# B&R Automation Studio project NAINV104C00R8L515F00 (part 37)

#### Act_OpsStandard_Hermes.st
```iecst
(** 2020-10-06 **)
ACTION Act_OpsStandard_Hermes:
	//InvertStepUSStandby
	//InvertStepAWMov
	IF eGotoOpsStep <> eOpsStep THEN

		CASE eGotoOpsStep OF

			ELSE
				eOpsStep	:= eGotoOpsStep;

		END_CASE

	END_IF

	Act_LogStep;

	IF eOpsStep = eGotoOpsStep THEN

		IF bPaused = FALSE THEN

			CASE eOpsStep OF

				InvertStepInitChkCondition:
					sStepTxt	:= 'Init Check Condition';

					IF p_bClampPrep THEN
						IF eInvertCurrPos	= InvertPosInvalid THEN
							bInvertPosInvalidSkipInit := TRUE;

							IF p_bClampDis THEN
								bClampDisInitUnblk	:= TRUE;
							END_IF

							eGotoOpsStep	:= InvertStepClampBlkBefInvert;
						ELSE
							eGotoOpsStep	:= InvertStepInitClampUnblk;
						END_IF
					ELSE
						IF eInvertCurrPos	= InvertPosInvalid THEN
							bInvertPosInvalidSkipInit := TRUE;

							IF (p_bInletShutterPrep AND p_bInletShutterDis=FALSE) OR (p_bOutletShutterPrep AND p_bOutletShutterDis=FALSE) THEN
								eGotoOpsStep	:= InvertStepShuttersCloseBefInvert;
							ELSE
								eGotoOpsStep	:= InvertStepInvert;
							END_IF
						ELSE
							eGotoOpsStep	:= InvertStepInitInvertComplChk;
						END_IF
					END_IF

					bPaused	:= p_bStop OR p_bStep;

				InvertStepInitClampUnblk:
					sStepTxt	:= 'Init Clamp Unblock';

					eClampAct	:= PneuActRet;

					IF p_eClampStatus = Done AND p_eClampStat = PneuActRet THEN

						eClampAct		:= PneuActIdle;
						eGotoOpsStep	:= InvertStepInitInvertComplChk;

						bPaused	:= p_bStop OR p_bStep;
					END_IF

				InvertStepInitInvertComplChk:
					sStepTxt	:= 'Init Checking Invert Complete Condition';

					IF bInvertCompl = FALSE THEN
						IF eInvertCurrPos = InvertCurrPosAtRemote THEN
							IF p_bLeftSen = TRUE THEN
								eGotoOpsStep	:= InvertStepInitConvAwayLftSen;
							ELSE
								eGotoOpsStep	:= InvertStepInitStopperBlk;
							END_IF

						ELSIF eInvertCurrPos = InvertCurrPosAtHome THEN
							IF p_bRightSen = TRUE THEN
								eGotoOpsStep	:= InvertStepInitConvAwayRgtSen;
							ELSE
								eGotoOpsStep	:= InvertStepInitStopperBlk;
							END_IF

						ELSE
							eGotoOpsStep	:= InvertStepInitStopperBlk;
						END_IF

					ELSE
						eGotoOpsStep	:= InvertStepInitStopperUnblk;
					END_IF

					bPaused	:= p_bStop OR p_bStep;

				InvertStepInitConvAwayLftSen:
					sStepTxt	:= 'Init Conveyor Away Stopper At Left';

					eConvAct	:= ConvActInit;

					fbFwdTimer(IN := TRUE, PT := DINT_TO_TIME(p_diFwdDlyTm));

					IF fbFwdTimer.Q = TRUE THEN
						fbFwdTimer(IN := FALSE);

						bHvBrd			:= FALSE;
						p_bConvHvBrd	:= FALSE;

						eConvAct		:= ConvActIdle;

						eGotoOpsStep	:= InvertStepInitStopperBlk;

						bPaused	:= p_bStop OR p_bStep;

					ELSIF p_eConvStatus = Done AND p_eConvStat = ConvActInit THEN
						fbFwdTimer(IN := FALSE);

						bHvBrd 			:= TRUE;
						bGdBrd			:= p_bInitGdBrd;

						eConvAct		:= ConvActIdle;

						eGotoOpsStep	:= InvertStepInitStopperBlk;

						bPaused	:= p_bStop OR p_bStep;
					END_IF

				InvertStepInitConvAwayRgtSen:
					sStepTxt	:= 'Init Conveyor Away Stopper At Right';

					eConvAct	:= ConvActRevImmedStart;

					fbRevTimer(IN := TRUE, PT := DINT_TO_TIME(p_diRevDlyTm));

					IF fbRevTimer.Q = TRUE THEN
						fbRevTimer(IN := FALSE);

						bHvBrd			:= FALSE;
						p_bConvHvBrd	:= FALSE;

						eConvAct		:= ConvActIdle;

						eGotoOpsStep	:= InvertStepInitStopperBlk;

						bPaused	:= p_bStop OR p_bStep;

					ELSIF p_eConvStatus = Done AND p_eConvStat = ConvActRevImmedStart THEN
						fbRevTimer(IN := FALSE);

						bHvBrd 			:= TRUE;
						bGdBrd			:= p_bInitGdBrd;

						eConvAct		:= ConvActIdle;

						eGotoOpsStep	:= InvertStepInitStopperBlk;

						bPaused	:= p_bStop OR p_bStep;
					END_IF

				InvertStepInitStopperBlk:
					sStepTxt	:= 'Init Stopper Block';

					eStopperAct	:= PneuActExt;

					IF p_eStopperStatus = Done AND p_eStopperStat = PneuActExt THEN
						eStopperAct := PneuActIdle;

						IF eInvertCurrPos = InvertCurrPosAtRemote THEN
							eGotoOpsStep  := InvertStepInitConvTwdLftSen;

						ELSIF eInvertCurrPos = InvertCurrPosAtHome THEN
							eGotoOpsStep  := InvertStepInitConvTwdRgtSen;
						END_IF

						bPaused	:= p_bStop OR p_bStep;
					END_IF

				InvertStepInitConvTwdLftSen:
					sStepTxt	:= 'Init Conveyor Toward Stopper At Left';

					eConvAct	:= ConvActRevImmedStart;

					fbRevTimer(IN := TRUE, PT := DINT_TO_TIME(p_diRevDlyTm));

					IF fbRevTimer.Q = TRUE THEN
						fbRevTimer(IN := FALSE);

						bHvBrd			:= FALSE;
						p_bConvHvBrd	:= FALSE;

						eConvAct		:= ConvActIdle;

						IF p_bClampPrep AND p_bClampDis=FALSE THEN
							eGotoOpsStep	:= InvertStepClampBlkBefInvert;
						ELSE
							IF (p_bInletShutterPrep AND p_bInletShutterDis=FALSE) OR (p_bOutletShutterPrep AND p_bOutletShutterDis=FALSE) THEN
								eGotoOpsStep	:= InvertStepShuttersCloseBefInvert;
							ELSE
								eGotoOpsStep	:= InvertStepInvert;
							END_IF
						END_IF

						bPaused	:= p_bStop OR p_bStep;

					ELSIF p_eConvStatus = Done AND p_eConvStat = ConvActRevImmedStart THEN
						fbRevTimer(IN := FALSE);
						eConvAct	:= ConvActIdle;

						bHvBrd			:= TRUE;
						bGdBrd			:= p_bInitGdBrd;

						IF p_bClampPrep AND p_bClampDis=FALSE THEN
							eGotoOpsStep	:= InvertStepClampBlkBefInvert;
						ELSE
							IF (p_bInletShutterPrep AND p_bInletShutterDis=FALSE) OR (p_bOutletShutterPrep AND p_bOutletShutterDis=FALSE) THEN
								eGotoOpsStep	:= InvertStepShuttersCloseBefInvert;
							ELSE
								eGotoOpsStep	:= InvertStepInvert;
							END_IF
						END_IF

						bPaused	:= p_bStop OR p_bStep;

					END_IF

				InvertStepInitConvTwdRgtSen:
					sStepTxt	:= 'Init Conveyor Toward Stopper at Right';

					eConvAct	:= ConvActInit;

					fbFwdTimer(IN := TRUE, PT := DINT_TO_TIME(p_diFwdDlyTm));

					IF fbFwdTimer.Q = TRUE THEN
						fbFwdTimer(IN := FALSE);

						bHvBrd			:= FALSE;
						p_bConvHvBrd	:= FALSE;

						eConvAct	:= ConvActIdle;

						IF p_bClampPrep AND p_bClampDis=FALSE THEN
							eGotoOpsStep	:= InvertStepClampBlkBefInvert;
						ELSE
							IF (p_bInletShutterPrep AND p_bInletShutterDis=FALSE) OR (p_bOutletShutterPrep AND p_bOutletShutterDis=FALSE) THEN
								eGotoOpsStep	:= InvertStepShuttersCloseBefInvert;
							ELSE
								eGotoOpsStep	:= InvertStepInvert;
							END_IF
						END_IF

						bPaused	:= p_bStop OR p_bStep;

					ELSIF p_eConvStatus = Done AND p_eConvStat = ConvActInit THEN
						fbFwdTimer(IN := FALSE);
						eConvAct	:= ConvActIdle;

						bHvBrd			:= TRUE;
						bGdBrd			:= p_bInitGdBrd;

						IF p_bClampPrep AND p_bClampDis=FALSE THEN
							eGotoOpsStep	:= InvertStepClampBlkBefInvert;
						ELSE
							IF (p_bInletShutterPrep AND p_bInletShutterDis=FALSE) OR (p_bOutletShutterPrep AND p_bOutletShutterDis=FALSE) THEN
								eGotoOpsStep	:= InvertStepShuttersCloseBefInvert;
							ELSE
								eGotoOpsStep	:= InvertStepInvert;
							END_IF
						END_IF

						bPaused	:= p_bStop OR p_bStep;
					END_IF

				InvertStepInitStopperUnblk:
					sStepTxt	:= 'Init Stopper Unblock';

					eStopperAct	:= PneuActRet;

					IF p_eStopperStatus = Done AND p_eStopperStat = PneuActRet THEN
						eStopperAct		:= PneuActIdle;
						eGotoOpsStep	:= InvertStepInitConvToRgt;

						bPaused	:= p_bStop OR p_bStep;
					END_IF

				InvertStepInitConvToRgt:
					sStepTxt	:= 'Init Conveyor to Right';

					eConvAct	:= ConvActInit;

					IF p_eConvStatus = Done AND p_eConvStat = ConvActInit THEN
						eConvAct		:= ConvActIdle;

						IF (p_bInletShutterPrep AND p_bInletShutterDis=FALSE) OR (p_bOutletShutterPrep AND p_bOutletShutterDis=FALSE) THEN
							eGotoOpsStep	:= InvertStepInitShuttersInOutClose;
						ELSE
							IF (p_bRightSen = TRUE AND NOT(p_bUSReversal)) OR (p_bLeftSen AND p_bUSReversal)   THEN //changed
								bHvBrd 	:= TRUE;
								bGdBrd	:= p_bInitGdBrd;

								eGotoOpsStep	:= InvertStepDSStandby;
							ELSE
								IF p_bAWWidthPosDiff = TRUE THEN
									eGotoOpsStep	:= InvertStepAWMov;
								ELSE
									eGotoOpsStep	:= InvertStepChkCondition;
								END_IF
							END_IF

						END_IF

						bPaused	:= p_bStop OR p_bStep;
					END_IF

				InvertStepInitShuttersInOutClose:
					sStepTxt			:= 'Init Closing Shutters';

					eInletShutterAct	:= PneuActExt;
					eOutletShutterAct	:= PneuActExt;

					IF (p_eInletShutterStatus = Done AND p_eInletShutterStat = PneuActExt) AND (p_eOutletShutterStatus = Done AND p_eOutletShutterStat = PneuActExt) THEN

						eInletShutterAct	:= PneuActIdle;
						eOutletShutterAct	:= PneuActIdle;

						IF (p_bRightSen = TRUE AND NOT(p_bUSReversal)) OR (p_bLeftSen AND p_bUSReversal)  THEN //changed

							bHvBrd 	:= TRUE;
							bGdBrd	:= p_bInitGdBrd;

							IF p_bOutletShutterOpen THEN
								eGotoOpsStep	:= InvertStepDSStandby;
							ELSE
								IF p_iHermesAction= 1 THEN
									eGotoOpsStep	:= InvertStepOutletShutterOpen;
								ELSE
									eGotoOpsStep	:= InvertStepDSInOutletShutterOpen;
								END_IF
							END_IF

						ELSE
							IF p_bAWWidthPosDiff = TRUE THEN
								eGotoOpsStep	:= InvertStepAWMov;
							ELSE
								eGotoOpsStep	:= InvertStepChkCondition;
							END_IF
						END_IF

						bPaused	:= p_bStop OR p_bStep;
					END_IF

				InvertStepShuttersInOutClose:
					sStepTxt			:= 'Closing Shutters Prior to Auto Width Change';

					eInletShutterAct	:= PneuActExt;
					eOutletShutterAct	:= PneuActExt;

					IF (p_eInletShutterStatus = Done AND p_eInletShutterStat = PneuActExt) AND (p_eOutletShutterStatus = Done AND p_eOutletShutterStat = PneuActExt) THEN

						eInletShutterAct	:= PneuActIdle;
						eOutletShutterAct	:= PneuActIdle;

						eGotoOpsStep	:= InvertStepAWMov;

						bPaused	:= p_bStop OR p_bStep;
					END_IF

				InvertStepAWMov:
					sStepTxt	:= 'Moving Auto Width';

					eAWAct	:= AWActGoWidthOff;

					IF (p_eAWStatus = Done AND p_eAWStat = AWActGoWidthOff) THEN
						eAWAct			:= AWActIdle;

						eGotoOpsStep	:= InvertStepChkCondition;

						bPaused	:= p_bStop OR p_bStep;
					END_IF

				InvertStepChkCondition:
					sStepTxt	:= 'Check Condition';

					IF (p_bInletShutterPrep AND p_bInletShutterDis=FALSE) OR (p_bOutletShutterPrep AND p_bOutletShutterDis=FALSE) THEN
						IF p_bUSAllow THEN
							eGotoOpsStep	:= InvertStepChkShutterCond;
						END_IF
					ELSE
						eGotoOpsStep	:= InvertStepStopperPosChk;
					END_IF

					bPaused	:= p_bStop OR p_bStep;

				InvertStepChkShutterCond:
					sStepTxt	:= 'Check Initial Shutter Condition';

					IF p_iHermesAction = 1 THEN
						IF p_bInletShutterOpen AND p_bOutletShutterOpen THEN//p_bOutletShutterClose THEN
							eGotoOpsStep:= InvertStepStopperPosChk;
						ELSE
							eGotoOpsStep:= InvertStepShuttersInOpenOutClose;
						END_IF
					ELSE
						IF p_bInletShutterOpen AND p_bOutletShutterOpen THEN
							eGotoOpsStep:= InvertStepStopperPosChk;
						ELSE
							eGotoOpsStep:= InvertStepShuttersInOutOpen;
						END_IF

					END_IF

					bPaused	:= p_bStop OR p_bStep;

					//Open both shutters if bypass mode
				InvertStepShuttersInOutOpen:
					sStepTxt			:= 'Opening Shutters Prior After Auto Width Change';

					eInletShutterAct	:= PneuActRet;
					eOutletShutterAct	:= PneuActRet;

					IF (p_eInletShutterStatus = Done AND p_eInletShutterStat = PneuActRet) AND (p_eOutletShutterStatus = Done AND p_eOutletShutterStat = PneuActRet) THEN

						eInletShutterAct	:= PneuActIdle;
						eOutletShutterAct	:= PneuActIdle;

						eGotoOpsStep	:= InvertStepStopperPosChk;

						bPaused	:= p_bStop OR p_bStep;
					END_IF

					//Open inlet shutter close outlet if invert mode
				InvertStepShuttersInOpenOutClose:
					sStepTxt			:= 'Opening Inlet Shutter and Closing Outlet Shutter';

					eInletShutterAct	:= PneuActRet;
					eOutletShutterAct	:= PneuActRet; //temporary testing

					IF (p_eInletShutterStatus = Done AND p_eInletShutterStat = PneuActRet) AND (p_eOutletShutterStatus = Done AND p_eOutletShutterStat = PneuActRet) THEN //PneuActExt

						eInletShutterAct	:= PneuActIdle;
						eOutletShutterAct	:= PneuActIdle;

						eGotoOpsStep	:= InvertStepStopperPosChk;

						bPaused	:= p_bStop OR p_bStep;
					END_IF

				InvertStepStopperPosChk:
					sStepTxt	:= 'Checking Stopper Position';

					IF eInvertCurrPos = InvertCurrPosAtRemote THEN
						IF NOT(p_iHermesAction = 1) THEN
							eGotoOpsStep	:= InvertStepStopperUnblk;
						ELSE
							IF NOT(p_bUSReversal) THEN
								eGotoOpsStep	:= InvertStepStopperUnblk;
							ELSE
								eGotoOpsStep	:= InvertStepStopperBlk;
							END_IF
						END_IF
					ELSIF eInvertCurrPos = InvertCurrPosAtHome THEN	//create condition if reversal
						IF NOT(p_iHermesAction = 1) THEN
							eGotoOpsStep	:= InvertStepStopperUnblk;
						ELSE
							IF NOT(p_bUSReversal) THEN
								eGotoOpsStep	:= InvertStepStopperBlk;
							ELSE
								eGotoOpsStep	:= InvertStepStopperUnblk;
							END_IF
						END_IF
					END_IF

					bPaused	:= p_bStop OR p_bStep;

				InvertStepStopperBlk:
					sStepTxt	:= 'Stopper Block';

					eStopperAct	:= PneuActExt;

					IF p_eStopperStatus = Done AND p_eStopperStat = PneuActExt THEN
						eStopperAct		:= PneuActIdle;
						eGotoOpsStep	:= InvertStepUSStandby;

						bPaused	:= p_bStop OR p_bStep;
					END_IF

				InvertStepStopperUnblk:
					sStepTxt	:= 'Stopper Unblock';

					eStopperAct	:= PneuActRet;

					IF p_eStopperStatus = Done AND p_eStopperStat = PneuActRet THEN
						eStopperAct		:= PneuActIdle;
						eGotoOpsStep	:= InvertStepUSStandby;

						bPaused	:= p_bStop OR p_bStep;
					END_IF

				InvertStepUSStandby:
					sStepTxt	:= 'In Upstream Standby Condition';

					bUSTimerRun	:= FALSE;

					bConvSen	:= p_bLeftSen OR p_bRightSen OR p_bMidSen;

					IF p_bAWWidthPosDiff = TRUE  THEN
						IF (p_bInletShutterPrep AND p_bInletShutterDis=FALSE) OR (p_bOutletShutterPrep AND p_bOutletShutterDis=FALSE) THEN
							eGotoOpsStep	:= InvertStepShuttersInOutClose;
						ELSE
							eGotoOpsStep	:= InvertStepAWMov;
						END_IF
					ELSIF p_bUSAllow = TRUE THEN
						eGotoOpsStep	:= InvertStepUSCommTmr;
					ELSIF bConvSen = TRUE THEN
						eGotoOpsStep	:= InvertStepUSTmr;
					END_IF

					bPaused	:= p_bStop OR p_bStep;

				InvertStepUSTmr:
					sStepTxt	:= 'Inserting Board By Timer';

					bConvSen	:= p_bLeftSen OR p_bRightSen OR p_bMidSen;

					fbUSTimer(IN := bConvSen);

					IF fbUSTimer.Q = TRUE THEN
						bUSTimerRun	:= TRUE;
						fbUSTimer(IN := FALSE);

						bGdBrd	:= p_bInsertGdBrd;

						IF p_iHermesAction = 1 THEN
							IF eInvertCurrPos = InvertCurrPosAtRemote THEN
								eGotoOpsStep	:= InvertStepEntToInOff;
							ELSIF eInvertCurrPos = InvertCurrPosAtHome THEN
								eGotoOpsStep	:= InvertStepEntToEnd;
							END_IF
						ELSE
							eGotoOpsStep	:= InvertStepEntToEnd;

						END_IF

					ELSIF bConvSen = FALSE THEN
						bUSTimerRun	:= FALSE;
						fbUSTimer(IN := FALSE);

						IF p_bAWWidthPosDiff = TRUE THEN
							IF (p_bInletShutterPrep AND p_bInletShutterDis=FALSE) OR (p_bOutletShutterPrep AND p_bOutletShutterDis=FALSE) THEN
								eGotoOpsStep	:= InvertStepShuttersInOutClose;
							ELSE
								eGotoOpsStep	:= InvertStepAWMov;
							END_IF
						ELSE
							eGotoOpsStep	:= InvertStepUSStandby;
						END_IF

					ELSE
						bPaused	:= p_bStop;

						IF bPaused = TRUE THEN
							bUSTimerRun	:= FALSE;
							fbUSTimer(IN := FALSE);

							eGotoOpsStep	:= InvertStepUSStandby;
						END_IF

					END_IF

				InvertStepUSCommTmr:
					sStepTxt	:= 'Communicating Upstream Machine';

					CASE p_eUSCommMod OF
						McSetCommModSMEMA:
							fbUSTimer(IN := p_bLeftSen OR p_bRightSen OR p_bMidSen);

							eUSSMEMAAct	:= SMEMAActRun;

							IF p_bUSSMEMATransporting = TRUE THEN
								bUSTimerRun	:= FALSE;
								fbUSTimer(IN := FALSE);

								bGdBrd			:= p_bUSSMEMAUSGdBrdRdy;

								sStepTxt		:= 'Conveyor Entering Board';

								IF p_iHermesAction = 1 THEN
									IF eInvertCurrPos = InvertCurrPosAtRemote THEN
										eGotoOpsStep	:= InvertStepEntToInOff;
									ELSIF eInvertCurrPos = InvertCurrPosAtHome THEN
										eGotoOpsStep	:= InvertStepEntToEnd;
									END_IF

								ELSE
									eGotoOpsStep	:= InvertStepEntToEnd;

								END_IF

							ELSIF fbUSTimer.Q = TRUE THEN
								bUSTimerRun	:= TRUE;
								fbUSTimer(IN := FALSE);

								bGdBrd	:= p_bInsertGdBrd;

								IF p_iHermesAction = 1 THEN
									IF eInvertCurrPos = InvertCurrPosAtRemote THEN
										eGotoOpsStep	:= InvertStepEntToInOff;
									ELSIF eInvertCurrPos = InvertCurrPosAtHome THEN
										eGotoOpsStep	:= InvertStepEntToEnd;
									END_IF
								ELSE
									eGotoOpsStep	:= InvertStepEntToEnd;
								END_IF

							ELSIF (p_bAWWidthPosDiff = TRUE) OR (p_bUSAllow = FALSE) THEN
								bUSTimerRun	:= FALSE;
								fbUSTimer(IN := FALSE);

								eUSSMEMAAct	:= SMEMAActIdle;

								IF p_bAWWidthPosDiff = TRUE THEN
									IF (p_bInletShutterPrep AND p_bInletShutterDis=FALSE) OR (p_bOutletShutterPrep AND p_bOutletShutterDis=FALSE) THEN
										eGotoOpsStep	:= InvertStepShuttersInOutClose;
									ELSE
										eGotoOpsStep	:= InvertStepAWMov;
									END_IF
								ELSE
									eGotoOpsStep	:= InvertStepUSStandby;
								END_IF

							ELSE

								bPaused	:= p_bStop;

								IF bPaused = TRUE THEN
									bUSTimerRun	:= FALSE;
									fbUSTimer(IN := FALSE);

									eUSSMEMAAct	:= SMEMAActIdle;

									eGotoOpsStep	:= InvertStepUSStandby;
								END_IF

							END_IF

						McSetCommModHermes:
							fbUSTimer(IN := p_bLeftSen OR p_bRightSen OR p_bMidSen);

							IF p_bUSHermesTransporting = TRUE  THEN
								bUSTimerRun	:= FALSE;
								fbUSTimer(IN := FALSE);

								bGdBrd	:= p_bUSHermesUSGdRdy;

								IF p_iHermesAction = 1 THEN
									IF eInvertCurrPos = InvertCurrPosAtRemote THEN
										IF NOT (p_bUSReversal) THEN
											eGotoOpsStep	:= InvertStepEntToInOff;
										ELSE
											eGotoOpsStep	:= InvertStepEntToEnd;
										END_IF
									ELSIF eInvertCurrPos = InvertCurrPosAtHome THEN
										IF NOT (p_bUSReversal) THEN
											eGotoOpsStep	:= InvertStepEntToEnd;
										ELSE
											eGotoOpsStep	:= InvertStepEntToInOff;
										END_IF
									END_IF
								ELSE //when bypass + reversal then check ds allow from which sided
									IF bReverseStoppingPos THEN
										eGotoOpsStep	:= InvertStepEntToInOff;
									ELSE
										eGotoOpsStep	:= InvertStepEntToEnd;
									END_IF
								END_IF

							ELSIF fbUSTimer.Q = TRUE THEN
								bUSTimerRun	:= TRUE;
								fbUSTimer(IN := FALSE);

								bGdBrd	:= p_bInsertGdBrd;

								IF p_iHermesAction = 1 THEN
									IF eInvertCurrPos = InvertCurrPosAtRemote THEN
										IF NOT (p_bUSReversal) THEN
											eGotoOpsStep	:= InvertStepEntToInOff;
										ELSE
											eGotoOpsStep	:= InvertStepEntToEnd;
										END_IF
									ELSIF eInvertCurrPos = InvertCurrPosAtHome THEN
										IF NOT (p_bUSReversal) THEN
											eGotoOpsStep	:= InvertStepEntToEnd;
										ELSE
											eGotoOpsStep	:= InvertStepEntToInOff;
										END_IF
									END_IF
								ELSE //when bypass + reversal then
									eGotoOpsStep	:= InvertStepEntToEnd;
								END_IF

							ELSIF (p_bAWWidthPosDiff = TRUE) OR (p_bUSAllow = FALSE) THEN
								bUSTimerRun	:= FALSE;
								fbUSTimer(IN := FALSE);

								IF p_bAWWidthPosDiff = TRUE THEN
									IF (p_bInletShutterPrep AND p_bInletShutterDis=FALSE) OR (p_bOutletShutterPrep AND p_bOutletShutterDis=FALSE) THEN
										eGotoOpsStep	:= InvertStepShuttersInOutClose;
									ELSE
										eGotoOpsStep	:= InvertStepAWMov;
									END_IF
								ELSE
									eGotoOpsStep	:= InvertStepUSStandby;
								END_IF

							ELSE

								bPaused	:= p_bStop;

								IF bPaused = TRUE THEN
									bUSTimerRun	:= FALSE;
									fbUSTimer(IN := FALSE);

									eGotoOpsStep	:= InvertStepUSStandby;
								END_IF

							END_IF

					END_CASE

				InvertStepEntToEnd:
					CASE p_eUSCommMod OF
						McSetCommModSMEMA:
							IF p_bUSSMEMATransporting = FALSE AND bUSTimerRun = FALSE THEN
								eConvAct	:= ConvActStop;

								IF p_eConvStatus = Done AND p_eConvStat = ConvActStop THEN
									eConvAct		:= ConvActIdle;

									eGotoOpsStep	:= InvertStepUSStandby;

									bPaused	:= p_bStop OR p_bStep;

								END_IF

							ELSE
								IF p_bUSSMEMAConvStart OR bUSTimerRun THEN
									sStepTxt	:= 'Conveyor Entering Board';
									eConvAct	:= ConvActEnt;
								END_IF

								IF (p_bConvHvBrd = TRUE) OR bUSTimerRun THEN
									bHvBrd := TRUE;
								END_IF

								IF p_bUSSMEMAConvStop AND bUSTimerRun = FALSE THEN
									sStepTxt	:= 'Conveyor Stopping';
									eConvAct	:= ConvActStop;
								END_IF

								//Waiting Conveyor Reach End for Invert Mode
								IF p_iHermesAction = 1 THEN
									IF ((p_eUSSMEMAStatus = Done AND p_eUSSMEMAStat = SMEMAActRun) OR (bUSTimerRun = TRUE)) AND p_eConvStatus = Done AND p_eConvStat = ConvActEnt THEN
										eUSSMEMAAct		:= SMEMAActIdle;
										eGotoOpsStep	:= InvertStepInvertComplChk;

										IF p_eConvStatus <> Busy THEN
											bPaused	:= p_bStop OR p_bStep;
										END_IF
									END_IF

								ELSE
									IF (p_eUSSMEMAStatus = Done AND p_eUSSMEMAStat = SMEMAActRun) OR (bUSTimerRun = TRUE) THEN
										eUSSMEMAAct		:= SMEMAActIdle;
										eGotoOpsStep	:= InvertStepInvertComplChk;

										IF p_eConvStatus <> Busy THEN
											bPaused	:= p_bStop OR p_bStep;
										END_IF
									END_IF

								END_IF

							END_IF

						McSetCommModHermes:
							IF p_bUSHermesTransporting  OR bUSTimerRun = TRUE THEN
								sStepTxt	:= 'Conveyor Entering Board';
								eConvAct	:= ConvActEnt;
							END_IF

							IF p_bUSHermesStopTransport = TRUE AND bUSTimerRun = FALSE THEN
								sStepTxt	:= 'Conveyor Stopping';
								eConvAct	:= ConvActStop;
							END_IF

							IF (p_bConvHvBrd = TRUE) OR (bUSTimerRun = TRUE) THEN
								bHvBrd := TRUE;
							END_IF

							//Waiting Conveyor Reach End for Invert Mode
							IF p_iHermesAction = 1 THEN
								IF p_bUSHermesTransporting = FALSE OR (bUSTimerRun) THEN
									IF p_eConvStat = ConvActStop THEN
										IF p_eConvStatus = Done THEN
											eConvAct		:= ConvActIdle;
											eGotoOpsStep	:= InvertStepUSStandby;
										END_IF
									ELSE
										IF p_eConvStatus = Done AND p_eConvStat = ConvActEnt THEN
											eGotoOpsStep	:= InvertStepInvertComplChk;
										END_IF
									END_IF

									IF p_eConvStatus <> Busy THEN
										bPaused	:= p_bStop OR p_bStep;
									END_IF
								END_IF

							ELSE
								IF p_bUSHermesTransporting = FALSE OR (bUSTimerRun) THEN
									IF p_eConvStat = ConvActStop THEN
										IF p_eConvStatus = Done THEN
											eConvAct		:= ConvActIdle;
											eGotoOpsStep	:= InvertStepUSStandby;
										END_IF
									ELSE
										eGotoOpsStep	:= InvertStepInvertComplChk;
									END_IF

									IF p_eConvStatus <> Busy THEN
										bPaused	:= p_bStop OR p_bStep;
									END_IF
								END_IF

							END_IF

					END_CASE

				InvertStepEntToInOff:
					CASE p_eUSCommMod OF
						McSetCommModSMEMA:
							IF p_bUSSMEMATransporting = FALSE AND bUSTimerRun = FALSE THEN
								eConvAct	:= ConvActStop;

								IF p_eConvStatus = Done AND p_eConvStat = ConvActStop THEN
									eConvAct		:= ConvActIdle;
									eGotoOpsStep	:= InvertStepUSStandby;

									bPaused	:= p_bStop OR p_bStep;

								END_IF

							ELSE
								IF p_bUSSMEMAConvStart OR bUSTimerRun THEN
									sStepTxt	:= 'Conveyor Entering Board';
									eConvAct	:= ConvActEntToInOff;
								END_IF

								IF (p_bConvHvBrd = TRUE) OR (bUSTimerRun = TRUE) THEN
									bHvBrd := TRUE;
								END_IF

								IF p_bUSSMEMAConvStop AND bUSTimerRun = FALSE THEN
									sStepTxt	:= 'Conveyor Stopping';
									eConvAct	:= ConvActStop;
								END_IF

								IF ((p_eUSSMEMAStatus = Done AND p_eUSSMEMAStat = SMEMAActRun) OR (bUSTimerRun = TRUE)) AND p_eConvStatus = Done AND p_eConvStat = ConvActEntToInOff THEN
									eUSSMEMAAct		:= SMEMAActIdle;
									eGotoOpsStep	:= InvertStepStopperBlkAftEnt;

									IF p_eConvStatus <> Busy THEN
										bPaused	:= p_bStop OR p_bStep;
									END_IF
								END_IF

							END_IF

						McSetCommModHermes:
							IF p_bUSHermesTransporting  OR bUSTimerRun = TRUE THEN
								sStepTxt	:= 'Conveyor Entering Board';
								eConvAct	:= ConvActEntToInOff;
							END_IF

							IF p_bUSHermesStopTransport = TRUE AND bUSTimerRun = FALSE THEN
								sStepTxt	:= 'Conveyor Stopping';
								eConvAct	:= ConvActStop;
							END_IF

							IF (p_bConvHvBrd = TRUE) OR (bUSTimerRun = TRUE) THEN
								bHvBrd	:= TRUE;
							END_IF

							IF (p_bUSHermesTransporting = FALSE  OR (bUSTimerRun)) THEN
								IF p_eConvStat = ConvActStop THEN
									IF p_eConvStatus = Done THEN
										eConvAct		:= ConvActIdle;
										eGotoOpsStep	:= InvertStepUSStandby;
									END_IF
								ELSE
									IF p_eConvStatus = Done AND p_eConvStat = ConvActEntToInOff THEN
										eGotoOpsStep	:= InvertStepStopperBlkAftEnt;
									END_IF
								END_IF

								IF p_eConvStatus <> Busy THEN
									bPaused	:= p_bStop OR p_bStep;
								END_IF
							END_IF

					END_CASE

				InvertStepStopperBlkAftEnt:
					sStepTxt	:= 'Stopper Block After Entering Board';

					eStopperAct	:= PneuActExt;

					IF p_eStopperStatus = Done AND p_eStopperStat = PneuActExt THEN
						eStopperAct		:= PneuActIdle;
						eGotoOpsStep	:= InvertStepRev;

						bPaused	:= p_bStop OR p_bStep;
					END_IF

				InvertStepRev:
					sStepTxt	:= 'Conveyor Reverse Board';

					eConvAct	:= ConvActRevImmedStart;

					IF p_eConvStatus = Done AND p_eConvStat = ConvActRevImmedStart THEN
						eConvAct		:= ConvActIdle;

						eGotoOpsStep	:= InvertStepInvertComplChk;

						bPaused	:= p_bStop OR p_bStep;
					END_IF

				InvertStepInvertComplChk:
					sStepTxt		:= 'Checking Invert Complete Condition';

					IF eInvertCurrPos <> eInvertReqPos THEN
						IF p_bClampPrep AND p_bClampDis=FALSE THEN
							eGotoOpsStep	:= InvertStepClampBlkBefInvert;
						ELSE
							IF (p_bInletShutterPrep AND p_bInletShutterDis=FALSE) OR (p_bOutletShutterPrep AND p_bOutletShutterDis=FALSE) THEN
								eGotoOpsStep	:= InvertStepShuttersCloseBefInvert;
							ELSE
								eGotoOpsStep	:= InvertStepInvert;
							END_IF
						END_IF
					ELSE
						IF (p_bInletShutterPrep AND p_bInletShutterDis=FALSE) OR (p_bOutletShutterPrep AND p_bOutletShutterDis=FALSE) THEN
							IF p_bOutletShutterOpen THEN
								eGotoOpsStep	:= InvertStepDSStandby;
							ELSE
								eGotoOpsStep	:= InvertStepOutletShutterOpen;
							END_IF
						ELSE //standby on right or left sensor ?
							eGotoOpsStep	:= InvertStepDSStandby;
						END_IF
					END_IF

					IF p_eConvStatus <> Busy THEN
						bPaused	:= p_bStop OR p_bStep;
					END_IF

				InvertStepClampBlkBefInvert:
					sStepTxt	:= 'Clamp Block Prior to Inversion';

					eClampAct	:= PneuActExt;

					IF p_eClampStatus = Done AND p_eClampStat = PneuActExt THEN

						eClampAct		:= PneuActIdle;

						IF (p_bInletShutterPrep AND p_bInletShutterDis=FALSE) OR (p_bOutletShutterPrep AND p_bOutletShutterDis=FALSE) THEN
							eGotoOpsStep	:= InvertStepShuttersCloseBefInvert;
						ELSE
							eGotoOpsStep	:= InvertStepInvert;
						END_IF

						bPaused	:= p_bStop OR p_bStep;
					END_IF

				InvertStepShuttersCloseBefInvert:
					sStepTxt			:= 'Closing Shutters Prior to Inversion';

					eInletShutterAct	:= PneuActExt;
					eOutletShutterAct	:= PneuActExt;

					IF (p_eInletShutterStatus = Done AND p_eInletShutterStat = PneuActExt) AND (p_eOutletShutterStatus = Done AND p_eOutletShutterStat = PneuActExt) THEN

						eInletShutterAct	:= PneuActIdle;
						eOutletShutterAct	:= PneuActIdle;

						eGotoOpsStep	:= InvertStepInvert;

						bPaused	:= p_bStop OR p_bStep;
					END_IF

				InvertStepInvert:
					sStepTxt	:= 'Inverter Turning';

					IF eInvertReqPos = InvertCurrPosAtRemote THEN
						eInvertAct	:= MotorBrkActCW;
					ELSIF eInvertReqPos = InvertCurrPosAtHome THEN
						eInvertAct	:= MotorBrkActCCW;
					END_IF

					IF p_eInvertStatus = Done AND (p_eInvertStat = MotorBrkActCW OR p_eInvertStat = MotorBrkActCCW)THEN
						eInvertAct		:= MotorBrkActIdle;

						IF (p_bClampPrep AND p_bClampDis=FALSE) OR bClampDisInitUnblk THEN

							bClampDisInitUnblk	:= FALSE;

							eGotoOpsStep	:= InvertStepClampUnblkAftInvert;

						ELSE
							IF eInvertCurrPos = InvertCurrPosAtRemote THEN

								IF bInvertPosInvalidSkipInit THEN
									eGotoOpsStep	:= InvertStepInvalidPosRecoverBrd;
								ELSE
									IF p_bLeftSen = TRUE THEN
										eGotoOpsStep	:= InvertStepPreExit;
									ELSE
										eGotoOpsStep	:= InvertStepChkCondition;
									END_IF
								END_IF

							ELSIF eInvertCurrPos = InvertCurrPosAtHome THEN

								IF bInvertPosInvalidSkipInit THEN
									eGotoOpsStep	:= InvertStepInvalidPosRecoverBrd;
								ELSE
									IF p_bRightSen = TRUE THEN
										eGotoOpsStep	:= InvertStepStopperUnblkAftInvert;
									ELSE
										eGotoOpsStep	:= InvertStepChkCondition;
									END_IF
								END_IF
							END_IF
						END_IF

						bPaused	:= p_bStop OR p_bStep;
					END_IF

				InvertStepClampUnblkAftInvert:
					sStepTxt	:= 'Clamp Unblock After Invert';

					eClampAct	:= PneuActRet;

					IF p_eClampStatus = Done AND p_eClampStat = PneuActRet THEN
						eClampAct		:= PneuActIdle;

						IF eInvertCurrPos = InvertCurrPosAtRemote THEN

							IF bInvertPosInvalidSkipInit THEN
								eGotoOpsStep	:= InvertStepInvalidPosRecoverBrd;
							ELSE
								IF p_bLeftSen = TRUE THEN
									eGotoOpsStep	:= InvertStepPreExit;
								ELSE
									eGotoOpsStep	:= InvertStepChkCondition;
								END_IF
							END_IF

						ELSIF eInvertCurrPos = InvertCurrPosAtHome THEN

							IF bInvertPosInvalidSkipInit THEN
								eGotoOpsStep	:= InvertStepInvalidPosRecoverBrd;
							ELSE
								IF p_bRightSen = TRUE THEN
									eGotoOpsStep	:= InvertStepStopperUnblkAftInvert;
								ELSE
									eGotoOpsStep	:= InvertStepChkCondition;
								END_IF
							END_IF
						END_IF

						bPaused	:= p_bStop OR p_bStep;

					END_IF

				InvertStepInvalidPosRecoverBrd:
					sStepTxt		:= 'Conveyor Recovering Board Status';

					eConvAct	:= ConvActInit;

					IF p_eConvStatus = Done AND p_eConvStat = ConvActInit THEN
						eConvAct		:= ConvActIdle;

						IF (p_bRightSen = TRUE AND NOT(p_bUSReversal)) OR (p_bLeftSen AND p_bUSReversal) THEN //changed
							bHvBrd := TRUE;
							bGdBrd			:= p_bInitGdBrd;

							bInvertPosInvalidSkipInit := FALSE;

							IF eInvertCurrPos = InvertCurrPosAtRemote THEN
								IF (p_bInletShutterPrep AND p_bInletShutterDis=FALSE) OR (p_bOutletShutterPrep AND p_bOutletShutterDis=FALSE) THEN
									IF p_bOutletShutterOpen THEN
										eGotoOpsStep	:= InvertStepDSStandby;
									ELSE
										eGotoOpsStep	:= InvertStepOutletShutterOpen;
									END_IF
								ELSE
									eGotoOpsStep	:= InvertStepDSStandby;
								END_IF
							ELSIF eInvertCurrPos = InvertCurrPosAtHome THEN
								eGotoOpsStep	:= InvertStepStopperUnblkAftInvert;
							END_IF

						ELSE
							bInvertPosInvalidSkipInit := FALSE;
							eGotoOpsStep	:= InvertStepChkCondition;
						END_IF

						bPaused	:= p_bStop OR p_bStep;
					END_IF

				InvertStepStopperUnblkAftInvert:
					sStepTxt	:= 'Stopper Unblock After Invert';

					eStopperAct	:= PneuActRet;

					IF p_eStopperStatus = Done AND p_eStopperStat = PneuActRet THEN
						eStopperAct		:= PneuActIdle;

						IF (p_bInletShutterPrep AND p_bInletShutterDis=FALSE) OR (p_bOutletShutterPrep AND p_bOutletShutterDis=FALSE) THEN
							IF p_bOutletShutterOpen THEN
								eGotoOpsStep	:= InvertStepDSStandby;
							ELSE
								eGotoOpsStep	:= InvertStepOutletShutterOpen;
							END_IF
						ELSE
							eGotoOpsStep	:= InvertStepDSStandby;
						END_IF

						bPaused	:= p_bStop OR p_bStep;
					END_IF

				InvertStepPreExit:
					sStepTxt		:= 'Conveyor Pre-Exiting Board';

					eConvAct	:= ConvActPreExit;

					IF p_eConvStatus = Done AND p_eConvStat = ConvActPreExit THEN
						eConvAct		:= ConvActIdle;

						IF (p_bInletShutterPrep AND p_bInletShutterDis=FALSE) OR (p_bOutletShutterPrep AND p_bOutletShutterDis=FALSE) THEN
							IF p_bOutletShutterOpen THEN
								eGotoOpsStep	:= InvertStepDSStandby;
							ELSE
								eGotoOpsStep	:= InvertStepOutletShutterOpen;
							END_IF
						ELSE
							eGotoOpsStep	:= InvertStepDSStandby;
						END_IF

						bPaused	:= p_bStop OR p_bStep;
					END_IF

				InvertStepDSInOutletShutterOpen:
					sStepTxt	:= 'DS: Opening Inlet & Outlet Shutter';

					eInletShutterAct	:= PneuActRet;
					eOutletShutterAct	:= PneuActRet;

					IF (p_eInletShutterStatus = Done AND p_eInletShutterStat = PneuActRet)
						AND (p_eOutletShutterStatus = Done AND p_eOutletShutterStat = PneuActRet)THEN

						eInletShutterAct	:= PneuActIdle;
						eOutletShutterAct	:= PneuActIdle;

						eGotoOpsStep	:= InvertStepDSStandby;

						bPaused	:= p_bStop OR p_bStep;
					END_IF

				InvertStepOutletShutterOpen:
					sStepTxt	:= 'Opening Outlet Shutter';

					eOutletShutterAct	:= PneuActRet;

					IF p_eOutletShutterStatus = Done AND p_eOutletShutterStat = PneuActRet THEN
						eOutletShutterAct	:= PneuActIdle;

						eGotoOpsStep	:= InvertStepDSStandby;

						bPaused	:= p_bStop OR p_bStep;
					END_IF

				InvertStepDSStandby:
					sStepTxt	:= 'In Downstream Standby Condition';

					bDSTimerRun	:= FALSE;

					IF p_bUSReversal THEN//p_eConvDirection = ConvDirLToL OR p_eConvDirection = ConvDirRToL THEN //tight with ds reversal
						bConvSen	:= p_bLeftSen;
					ELSE
						bConvSen	:= p_bRightSen;
					END_IF

					IF bConvSen = TRUE OR p_eConvStatus <> Busy THEN
						bReachedEnd	:= TRUE;
					END_IF

					IF p_bDBAOnRgtSen THEN
						IF p_bDSAllow = TRUE AND bReachedEnd = TRUE THEN
							bReachedEnd		:= FALSE;
							eGotoOpsStep	:= InvertStepDSCommTmr;
						ELSIF (bReachedEnd = TRUE) AND (bConvSen = FALSE) THEN
							bReachedEnd		:= FALSE;
							eGotoOpsStep	:= InvertStepDSTmr;
						END_IF
					ELSE
						IF p_bDSAllow = TRUE THEN
							bReachedEnd		:= FALSE;
							eGotoOpsStep	:= InvertStepDSCommTmr;
						ELSIF (bReachedEnd = TRUE) AND (bConvSen = FALSE) THEN
							bReachedEnd		:= FALSE;
							eGotoOpsStep	:= InvertStepDSTmr;
						END_IF
					END_IF

					IF p_eConvStatus <> Busy THEN
						bPaused	:= p_bStop OR p_bStep;
					END_IF

				InvertStepDSTmr:
					sStepTxt	:= 'Removing Board By Timer';

					IF p_bUSReversal THEN// p_eConvDirection = ConvDirLToL OR p_eConvDirection = ConvDirRToL THEN
						bConvSen	:= p_bLeftSen;
					ELSE
						bConvSen	:= p_bRightSen;
					END_IF

					fbDSTimer(IN := NOT bConvSen);

					IF fbDSTimer.Q = TRUE THEN
						bDSTimerRun		:= TRUE;
						fbDSTimer(IN := FALSE);

						bHvBrd := FALSE;

						eConvAct		:= ConvActIdle;

						eGotoOpsStep	:= InvertStepChkCondition;

					ELSIF bConvSen = TRUE THEN
						bDSTimerRun		:= FALSE;
						fbDSTimer(IN := FALSE);

						eGotoOpsStep	:= InvertStepDSStandby;

					ELSE
						IF p_eConvStatus <> Busy THEN
							bPaused	:= p_bStop;

							IF bPaused = TRUE THEN
								bDSTimerRun	:= FALSE;
								fbDSTimer(IN := FALSE);
							END_IF
						END_IF

					END_IF

				InvertStepDSCommTmr:
					sStepTxt	:= 'Communicating Downstream Machine';

					IF p_bUSReversal THEN// p_eConvDirection = ConvDirLToL OR p_eConvDirection = ConvDirRToL THEN
						IF p_bLeftSen = TRUE OR p_eConvStatus <> Busy THEN
							bReachedEnd	:= TRUE;
						END_IF

						IF bReachedEnd = TRUE THEN
							fbDSTimer(IN := NOT p_bLeftSen);
						END_IF
					ELSE
						IF p_bRightSen = TRUE OR p_eConvStatus <> Busy THEN
							bReachedEnd	:= TRUE;
						END_IF

						IF bReachedEnd = TRUE THEN
							fbDSTimer(IN := NOT p_bRightSen);
						END_IF
					END_IF

					CASE p_eDSCommMod OF
						McSetCommModSMEMA:
							eDSSMEMAAct	:= SMEMAActRun;

							IF p_bDSSMEMAConvStart = TRUE THEN
								bDSTimerRun	:= FALSE;
								fbDSTimer(IN := FALSE);

								bReachedEnd	:= FALSE;

								eGotoOpsStep	:= InvertStepExitBrd;

							ELSIF fbDSTimer.Q = TRUE THEN
								bDSTimerRun		:= TRUE;
								fbDSTimer(IN := FALSE);
								bHvBrd := FALSE;

								bReachedEnd		:= FALSE;
								eDSSMEMAAct		:= SMEMAActIdle;
								eConvAct		:= ConvActIdle;

								eGotoOpsStep	:= InvertStepChkCondition;

							ELSIF p_bDSAllow = FALSE THEN
								bDSTimerRun		:= FALSE;
								fbDSTimer(IN := FALSE);

								bReachedEnd		:= FALSE;
								eDSSMEMAAct		:= SMEMAActIdle;
								eConvAct		:= ConvActIdle;

								eGotoOpsStep	:= InvertStepDSStandby;

							ELSE
								IF p_eConvStatus <> Busy THEN
									bPaused	:= p_bStop;

									IF bPaused = TRUE THEN
										fbDSTimer(IN := FALSE);

										eDSSMEMAAct	:= SMEMAActIdle;
									END_IF
								END_IF

							END_IF

						McSetCommModHermes:
							IF p_bDSHermesTransporting = TRUE THEN
								bDSTimerRun	:= FALSE;
								fbDSTimer(IN := FALSE);

								bReachedEnd	:= FALSE;

								eGotoOpsStep	:= InvertStepExitBrd;

							ELSIF fbDSTimer.Q = TRUE THEN
								bDSTimerRun	:= TRUE;
								fbDSTimer(IN := FALSE);
								bHvBrd := FALSE;

								bReachedEnd	:= FALSE;
								eConvAct		:= ConvActIdle;

								eGotoOpsStep	:= InvertStepChkCondition;

							ELSIF p_bDSAllow = FALSE THEN
								bDSTimerRun	:= FALSE;
								fbDSTimer(IN := FALSE);

								bReachedEnd	:= FALSE;

								eGotoOpsStep	:= InvertStepDSStandby;

							ELSE
								IF p_eConvStatus <> Busy THEN
									bPaused	:= p_bStop;

									IF bPaused = TRUE THEN
										fbDSTimer(IN := FALSE);
									END_IF
								END_IF

							END_IF

					END_CASE

				InvertStepExitBrd:
					CASE p_eDSCommMod OF
						McSetCommModSMEMA:
							eConvAct	:= ConvActExit;

							IF ((p_eDSSMEMAStatus = Done AND p_eDSSMEMAStat = SMEMAActRun) OR (bDSTimerRun)) AND (p_eConvStatus = Done AND p_eConvStat = ConvActExit) THEN

								eDSSMEMAAct		:= SMEMAActIdle;
								eConvAct		:= ConvActIdle;

								bHvBrd := FALSE;
								p_bConvHvBrd := FALSE;
								eGotoOpsStep	:= InvertStepChkCondition;

								bPaused	:= p_bStop OR p_bStep;

							END_IF

						McSetCommModHermes:
							eConvAct := ConvActExit;

							IF ((p_bDSHermesTransporting = FALSE) OR (bDSTimerRun)) AND (p_eConvStatus = Done AND p_eConvStat = ConvActExit) THEN
								eConvAct := ConvActIdle;

								bHvBrd := FALSE;
								p_bConvHvBrd := FALSE;

								eGotoOpsStep := InvertStepChkCondition;

								bPaused := p_bStop OR p_bStep;
							END_IF

					END_CASE

			END_CASE

		END_IF

	END_IF

	//Board Inserted/Removed
	bBrdInserted		:= bUSTimerRun;
	bBrdRemoved			:= bDSTimerRun;

	//Operation Step Status
	IF (eOpsStep = InvertStepInitConvAwayLftSen) OR (eOpsStep = InvertStepInitConvAwayRgtSen) OR (eOpsStep = InvertStepInitConvTwdLftSen) OR (eOpsStep = InvertStepInitConvTwdRgtSen) OR (eOpsStep = InvertStepInitConvToRgt) THEN
		bStepInitConv	:= TRUE;
	ELSE
		bStepInitConv	:= FALSE;
	END_IF

	bStepInitAwayStopper		:= (eOpsStep = InvertStepInitConvAwayLftSen) OR (eOpsStep = InvertStepInitConvAwayRgtSen);
	bStepInitTwdStopper			:= (eOpsStep = InvertStepInitConvTwdLftSen) OR (eOpsStep = InvertStepInitConvTwdRgtSen);
	bStepInitDone				:= (eOpsStep > InvertStepInitShuttersInOutClose) AND bInvertPosInvalidSkipInit=FALSE;
	bStepUSStandby				:= eOpsStep = InvertStepUSStandby;
	bStepUSCommTmr				:= eOpsStep = InvertStepUSCommTmr;
	bStepEntToEnd				:= eOpsStep = InvertStepEntToEnd;
	bStepEntToInOff				:= eOpsStep = InvertStepEntToInOff;
	bStepRev					:= eOpsStep = InvertStepRev;
	bStepPreExit				:= eOpsStep = InvertStepPreExit;
	bStepDSStandby				:= eOpsStep = InvertStepDSStandby;
	bStepDSCommTmr				:= eOpsStep = InvertStepDSCommTmr;
	bStepExitBrd				:= eOpsStep = InvertStepExitBrd;
	bStepInvert					:= eOpsStep = InvertStepInvert;
	bStepAWMov					:= eOpsStep = InvertStepAWMov;
END_ACTION
```

#### InputRef.var - Do Not Change!!!
```iecst
(*2020-10-06*)
(**)
(*General*)
VAR
	p_udiRstErr : REFERENCE TO UDINT;
	p_bEn : REFERENCE TO BOOL;
	p_bDis : REFERENCE TO BOOL;
	p_bRun : REFERENCE TO BOOL;
	p_bStop : REFERENCE TO BOOL;
	p_bStep : REFERENCE TO BOOL;
END_VAR
(**)
VAR
	p_bInitGdBrd : REFERENCE TO BOOL;
	p_bInsertGdBrd : REFERENCE TO BOOL;
	p_eConvDirection : REFERENCE TO eConvDir;
	p_eUSCommMod : REFERENCE TO eMcSetCommMod;
	p_eDSCommMod : REFERENCE TO eMcSetCommMod;
	p_bGoToStandby : REFERENCE TO BOOL;
	p_bUSAllow : REFERENCE TO BOOL;
	p_bDSAllow : REFERENCE TO BOOL;
	p_eUSComm2Mod : REFERENCE TO eMcSetCommMod;
	p_bRtrnUSAllow : REFERENCE TO BOOL;
	p_bRtrnDSAllow : REFERENCE TO BOOL;
	p_bLeftSen : REFERENCE TO BOOL;
	p_bRightSen : REFERENCE TO BOOL;
	p_bMidSen : REFERENCE TO BOOL;
	p_bClamp2Sen : REFERENCE TO BOOL;
	p_bClamp3Sen : REFERENCE TO BOOL;
END_VAR
(**)
VAR
	p_eUSSMEMAStat : REFERENCE TO eSMEMAAction;
	p_eUSSMEMAStatus : REFERENCE TO eFBStatus;
	p_bUSSMEMATransporting : REFERENCE TO BOOL;
	p_bUSSMEMAConvStart : REFERENCE TO BOOL;
	p_bUSSMEMAConvStop : REFERENCE TO BOOL;
	p_bUSSMEMAUSRdy : REFERENCE TO BOOL;
	p_bUSSMEMAUSGdBrdRdy : REFERENCE TO BOOL;
END_VAR
(**)
VAR
	p_eUSSMEMA2Stat : REFERENCE TO eSMEMAAction;
	p_eUSSMEMA2Status : REFERENCE TO eFBStatus;
	p_bUSSMEMA2Transporting : REFERENCE TO BOOL;
	p_bUSSMEMA2ConvStart : REFERENCE TO BOOL;
	p_bUSSMEMA2ConvStop : REFERENCE TO BOOL;
	p_bUSSMEMA2USRdy : REFERENCE TO BOOL;
	p_bUSSMEMA2USGdBrdRdy : REFERENCE TO BOOL;
END_VAR
(**)
VAR
	p_eDSSMEMAStat : REFERENCE TO eSMEMAAction;
	p_eDSSMEMAStatus : REFERENCE TO eFBStatus;
	p_bDSSMEMAConvStart : REFERENCE TO BOOL;
	p_bDSSMEMAConvStop : REFERENCE TO BOOL;
	p_bDSSMEMATimer : REFERENCE TO BOOL;
	p_bDBAOnRgtSen : REFERENCE TO BOOL;
END_VAR
(**)
VAR
	p_bUSHermesTransporting : REFERENCE TO BOOL;
	p_bUSHermesStopTransport : REFERENCE TO BOOL;
	p_bUSHermesUSRdy : REFERENCE TO BOOL;
	p_bUSHermesUSGdRdy : REFERENCE TO BOOL;
END_VAR
(**)
VAR
	p_bDSHermesTransporting : REFERENCE TO BOOL;
	p_bDSHermesStopTransport : REFERENCE TO BOOL;
END_VAR
(**)
VAR
	p_eConvStat : REFERENCE TO eConvAction;
	p_eConvStatus : REFERENCE TO eFBStatus;
	p_bConvHvBrd : REFERENCE TO BOOL;
END_VAR
(**)
VAR
	p_eStopperStat : REFERENCE TO ePneuAction;
	p_eStopperStatus : REFERENCE TO eFBStatus;
	p_bStopperExtended : REFERENCE TO BOOL;
	p_bStopperRetracted : REFERENCE TO BOOL;
END_VAR
(**)
VAR
	p_eClampStat : REFERENCE TO ePneuAction;
	p_eClampStatus : REFERENCE TO eFBStatus;
END_VAR
(**)
VAR
	p_eInletShutterStat : REFERENCE TO ePneuAction;
	p_eInletShutterStatus : REFERENCE TO eFBStatus;
	p_bInletShutterOpen : REFERENCE TO BOOL;
	p_bInletShutterClose : REFERENCE TO BOOL;
END_VAR
(**)
VAR
	p_eOutletShutterStat : REFERENCE TO ePneuAction;
	p_eOutletShutterStatus : REFERENCE TO eFBStatus;
	p_bOutletShutterOpen : REFERENCE TO BOOL;
	p_bOutletShutterClose : REFERENCE TO BOOL;
END_VAR
(**)
VAR
	p_eClamp1Stat : REFERENCE TO ePneuAction;
	p_eClamp1Status : REFERENCE TO eFBStatus;
	p_bClampRS1 : REFERENCE TO BOOL;
	p_bUnClampRS1 : REFERENCE TO BOOL;
END_VAR
(**)
VAR
	p_eClamp2Stat : REFERENCE TO ePneuAction;
	p_eClamp2Status : REFERENCE TO eFBStatus;
	p_bClampRS2 : REFERENCE TO BOOL;
	p_bUnClampRS2 : REFERENCE TO BOOL;
END_VAR
(**)
VAR
	p_eClamp3Stat : REFERENCE TO ePneuAction;
	p_eClamp3Status : REFERENCE TO eFBStatus;
	p_bClampRS3 : REFERENCE TO BOOL;
	p_bUnClampRS3 : REFERENCE TO BOOL;
END_VAR
(**)
VAR
	p_eInvertStat : REFERENCE TO eMotorBrkAction;
	p_eInvertStatus : REFERENCE TO eFBStatus;
END_VAR
(**)
VAR
	p_eAWStat : REFERENCE TO eAWAction;
	p_eAWStatus : REFERENCE TO eFBStatus;
	p_bAWWidthPosDiff : REFERENCE TO BOOL;
END_VAR
(**)
VAR
	p_sProgNm : REFERENCE TO STRING[15];
	p_bNtSettingsLoadDone : REFERENCE TO BOOL;
END_VAR
(**)
VAR
	p_bClampPrep : REFERENCE TO BOOL;
	p_bClampDis : REFERENCE TO BOOL;
	p_eClampOption : REFERENCE TO eClampType;
END_VAR
(**)
VAR
	p_bInletShutterPrep : REFERENCE TO BOOL;
	p_bInletShutterDis : REFERENCE TO BOOL;
	p_bOutletShutterPrep : REFERENCE TO BOOL;
	p_bOutletShutterDis : REFERENCE TO BOOL;
END_VAR
(**)
VAR
	p_bMachineSafetyPrep : REFERENCE TO BOOL;
	p_bUnlockCovPrep : REFERENCE TO BOOL;
	p_bLinkDICoverSwitchSig2 : REFERENCE TO BOOL;
	p_bLinkUIBypsCoverSWPress1 : REFERENCE TO BOOL;
	p_bLinkDIUnlockCoverSigFromDS : REFERENCE TO BOOL;
	p_bLinkDISafetySigFromDS : REFERENCE TO BOOL;
	p_bLinkDISafetySigFromUS : REFERENCE TO BOOL;
	p_bLinkDIUnlockCoverSigFromUS : REFERENCE TO BOOL;
END_VAR
(*Route Action Hermes Operaiton*)
VAR
	p_iHermesAction : REFERENCE TO INT;
	p_bUSReversal : REFERENCE TO BOOL;
	p_bHermesEntToReversePosition : REFERENCE TO BOOL;
END_VAR
```

#### Local.var - Do Not Change!!!
```iecst
(*2020-10-06*)
(**)
(*Local Action, State & Status*)
VAR
	eStatus : eFBStatus := Idle;
	udiStatus : UDINT := 0;
	udiStatus1 : UDINT := 0;
END_VAR
(**)
(*Local Alarm*)
VAR
	tyAlmData : tyAlmDat;
	tyAlmData1 : tyAlmDat;
	a_tyAlmText : ARRAY[10000..10099] OF tyAlmTxt := [9(0),(sAlmText:='Waiting for Return PCB from Upstream 2'),(sAlmText:='Waiting for Return PCB Transfer to Downstream'),89(0)];
END_VAR
(**)
(*Local Output*)
VAR
	sStepTxt : STRING[80];
	bPaused : BOOL;
END_VAR
(**)
VAR
	bStepInitConv : BOOL;
	bStepInitAwayStopper : BOOL;
	bStepInitTwdStopper : BOOL;
	bStepInitDone : BOOL;
	bStepUSStandby : BOOL;
	bStepUSCommTmr : BOOL;
	bStepEntToEnd : BOOL;
	bStepEntToInOff : BOOL;
	bStepRev : BOOL;
	bStepPreExit : BOOL;
	bStepDSStandby : BOOL;
	bStepDSCommTmr : BOOL;
	bStepExitBrd : BOOL;
	bStepInvert : BOOL;
	bStepAWMov : BOOL;
	bStepSafeMode : BOOL;
	bBrdInserted : BOOL;
	bBrdRemoved : BOOL;
	eUSSMEMAAct : eSMEMAAction;
	eDSSMEMAAct : eSMEMAAction;
	eUSSMEMA2Act : eSMEMAAction;
	eConvAct : eConvAction;
	eStopperAct : ePneuAction;
	eInvertAct : eMotorBrkAction;
	eAWAct : eAWAction;
	eClampAct : ePneuAction;
	eInletShutterAct : ePneuAction;
	eOutletShutterAct : ePneuAction;
	eClamp1Act : ePneuAction;
	eClamp2Act : ePneuAction;
	eClamp3Act : ePneuAction;
	bInvOnceTwicePCBOut : BOOL;
	bStepInvRtrnEntToEnd : BOOL;
	bStepInvRtrnEntToInOff : BOOL;
	bStepInvRtrnUSStandby : BOOL;
	bStepInvRtrnUSCommTmr : BOOL;
END_VAR
(**)
(*Local Input*)
VAR
	udiRstErr : UDINT := 0;
	bEn : BOOL := TRUE;
	bDis : BOOL := FALSE;
	bRun : BOOL;
	bStop : BOOL;
	bStep : BOOL;
	bInletShutterPrep : BOOL;
	bInletShutterDis : BOOL;
	bOutletShutterPrep : BOOL;
	bOutletShutterDis : BOOL;
	bClampPrep : BOOL;
	bClampDis : BOOL;
	eClampOption : eClampType;
END_VAR
(**)
VAR
	bBrdOnSen : BOOL := FALSE;
	bHvBrd : BOOL;
	bGdBrd : BOOL;
	bInitGdBrd : BOOL := TRUE;
	bInsertGdBrd : BOOL := TRUE;
	eConvDirection : eConvDir;
	eUSCommMod : eMcSetCommMod;
	eDSCommMod : eMcSetCommMod;
	bGoToStandby : BOOL;
	bUSAllow : BOOL := TRUE;
	bDSAllow : BOOL := TRUE;
	bLeftSen : BOOL;
	bRightSen : BOOL;
	bMidSen : BOOL;
	bClamp2Sen : BOOL;
	bClamp3Sen : BOOL;
	bRtrnUSAllow : BOOL := TRUE;
	bRtrnDSAllow : BOOL := TRUE;
END_VAR
(**)
VAR
	eUSSMEMAStat : eSMEMAAction;
	eUSSMEMAStatus : eFBStatus;
	bUSSMEMATransporting : BOOL;
	bUSSMEMAConvStart : BOOL;
	bUSSMEMAConvStop : BOOL;
	bUSSMEMAUSRdy : BOOL;
	bUSSMEMAUSGdBrdRdy : BOOL;
END_VAR
(**)
VAR
	eDSSMEMAStat : eSMEMAAction;
	eDSSMEMAStatus : eFBStatus;
	bDSSMEMAConvStart : BOOL;
	bDSSMEMAConvStop : BOOL;
	bDSSMEMATimer : BOOL;
END_VAR
(**)
VAR
	bUSHermesTransporting : BOOL;
	bUSHermesStopTransport : BOOL;
	bUSHermesUSRdy : BOOL;
	bUSHermesUSGdRdy : BOOL;
END_VAR
(**)
VAR
	bDSHermesTransporting : BOOL;
	bDSHermesStopTransport : BOOL;
END_VAR
(**)
VAR
	eConvStat : eConvAction;
	eConvStatus : eFBStatus;
	bConvHvBrd : BOOL;
	bConvLmtSenActivated : BOOL;
END_VAR
(**)
VAR
	eStopperStat : ePneuAction;
	eStopperStatus : eFBStatus;
	bStopperExtended : BOOL;
	bStopperRetracted : BOOL;
END_VAR
(**)
VAR
	eClampStat : ePneuAction;
	eClampStatus : eFBStatus;
END_VAR
(**)
VAR
	eInletShutterStat : ePneuAction;
	eInletShutterStatus : eFBStatus;
	bInletShutterClose : BOOL;
	bInletShutterOpen : BOOL;
	eOutletShutterStat : ePneuAction;
	eOutletShutterStatus : eFBStatus;
	bOutletShutterClose : BOOL;
	bOutletShutterOpen : BOOL;
END_VAR
(**)
VAR
	eClamp1Stat : ePneuAction;
	eClamp1Status : eFBStatus;
	bClampRS1 : BOOL;
	bUnClampRS1 : BOOL;
END_VAR
(**)
VAR
	eClamp2Stat : ePneuAction;
	eClamp2Status : eFBStatus;
	bClampRS2 : BOOL;
	bUnClampRS2 : BOOL;
END_VAR
(**)
VAR
	eClamp3Stat : ePneuAction;
	eClamp3Status : eFBStatus;
	bClampRS3 : BOOL;
	bUnClampRS3 : BOOL;
END_VAR
(**)
VAR
	sProgNm : STRING[15] := 'Ops Conv';
	bNtSettingsLoadDone : BOOL := TRUE;
END_VAR
(**)
VAR
	diFwdDlyTm : DINT := 5000;
	diRevDlyTm : DINT := 5000;
END_VAR
(**)
(*Local*)
VAR
	bRstErr : BOOL;
	udiRstErrOld : UDINT;
	bInitDone : BOOL;
	bInitialDone : BOOL;
	eOpsStep : eInvertStep := InvertStepNA;
	eGotoOpsStep : eInvertStep := InvertStepInitChkCondition;
	fbUSTimer : TON := (PT:=T#1s);
	fbDSTimer : TON := (PT:=T#1s);
	bUSTimerRun : BOOL;
	bDSTimerRun : BOOL;
	fbUS2Timer : TON := (PT:=T#1s);
	bUS2TimerRun : BOOL;
	bConvSen : BOOL;
	bReachedEnd : BOOL;
	fbFwdTimer : TON;
	fbRevTimer : TON;
	bInvertPosInvalidSkipInit : BOOL;
	bClampDisInitUnblk : BOOL;
	bChangeBypassRetPneu : BOOL;
	bChangeInvertExtPneu : BOOL;
	bBoardInFromUS1 : BOOL;
	bBoardInFromUS2 : BOOL;
	bReverseStoppingPos : BOOL;
	udiModuleNum : UDINT := 6051;
END_VAR
(*Step Logger*)
VAR
	bClsLog : BOOL;
	blog : BOOL;
	logStep : ARRAY[0..999] OF eInvertStep;
	logIndexStep : INT;
	eGotoOpsStepDummy : eInvertStep;
	btest : BOOL;
END_VAR
```

### Machine.var - Change By Project
```iecst
(*2018-12-07*)
(**)
(*Action & State & Status*)
(**)
(*Alarm*)
VAR
	p_McAlmData : UDINT;
	p_McAlmData1 : UDINT;
END_VAR
(**)
(*Output*)
```

### Program Logical/Machine/Machine (IEC, version 1.00.0) - 1.00.0 - 

#### Init.st - Change By Project
```iecst
(** 2019-03-22 **)
PROGRAM _INIT

	(* Always Change If Project Change *)

	//Pass Address To Global Address For External Use
	//Action, State & Status

	//Alarm
	p_McAlmData		:= ADR(tyAlmData);
	p_McAlmData1	:= ADR(tyAlmData1);

	//Output

	(* Always Change If Project Change *)

END_PROGRAM
```

#### Act_InitGlobal.st - Change By Project
```iecst
(** 2019-04-09 **)
ACTION Act_InitGlobal:

	(* Always Change If Project Change *)

	//Pass Data To Link

	//Pass Data To Internal Use
	p_udiRstErr ACCESS p_RstErrReset;

	p_bOpsRun ACCESS p_OpsRun;
	p_bDIThermalPrtSig ACCESS p_DIThermalPrtSig;
	p_bDIPressureSW ACCESS p_DIPressureSW;

	p_sProgNm ACCESS p_NtParamMcProgNm;
	p_bNtSettingsLoadDone ACCESS p_StartupNtSettingsLoadDone;

	p_tyNtParamCurr ACCESS p_NtParamCurr;

	(* Always Change If Project Change *)

END_ACTION
```

#### Cyclic.st - Change By Project
```iecst
(** 2019-03-22 **)
PROGRAM _CYCLIC

	IF bInitDone = FALSE THEN
		bInitDone	:= TRUE;

		Act_InitLocal;
		Act_InitGlobal;

	ELSIF bInitialDone = FALSE THEN
		IF p_bNtSettingsLoadDone = TRUE THEN
			bInitialDone	:= TRUE;

			Act_Initial;
		END_IF

	ELSE

		Act_RstErr;
		Act_Background;
		Act_Alarm;
		//Act_AlarmInfo;
		Act_Alarm1;

	END_IF

END_PROGRAM
```

#### Act_InitLocal.st - Change By Project
```iecst
(** 2020-10-06 **)
ACTION Act_InitLocal:

	//Input Reference Link To Local Variable
	p_udiRstErr ACCESS ADR(udiRstErr);
	p_sProgNm ACCESS ADR(sProgNm);
	p_bNtSettingsLoadDone ACCESS ADR(bNtSettingsLoadDone);

	p_bDIThermalPrtSig ACCESS ADR(bThermalPrtSig);
	p_bDIPressureSW ACCESS ADR(bPressureSW);

	p_tyNtParamCurr ACCESS ADR(tyNtParamCurr);

END_ACTION
```

#### Act_Initial.st - Change By Project
```iecst
(** 2018-12-07 **)
ACTION Act_Initial:

	//Initial

END_ACTION
```

#### Act_Background.st - Change By Project
```iecst
(** 2020-10-08 **)
ACTION Act_Background:

//	Thermal Signal
	IF (p_bOpsRun = TRUE AND p_bDIThermalPrtSig = FALSE AND p_tyNtParamCurr.tyDISettings.diThermalPrtSig<>0) AND (eStatus <> Error) THEN
		eStatus		:= Error;
		udiStatus	:= 10001;	//Thermal Protection Signal Not Activated
	END_IF

	IF (p_bOpsRun = TRUE AND p_bDIPressureSW = FALSE AND p_tyNtParamCurr.tyDISettings.diPressureSW<>0) AND (eStatus <> Error) THEN
		eStatus		:= Error;
		udiStatus	:= 10000;	//Pressure Switch Not Activated
	END_IF

//Reset Error
	IF (eStatus = Error) AND bRstErr THEN
		eStatus		:= Idle;
		udiStatus	:= 0;
	END_IF

END_ACTION
```

#### Act_Alarm.st - Change By Project
```iecst
(** 2019-03-25 **)
ACTION Act_Alarm:

	//Error
	IF EDGEPOS(eStatus = Error) THEN

		tyAlmData.sProgNm		:= p_sProgNm;
		tyAlmData.udiCode		:= udiStatus;
		tyAlmData.eSeverity		:= AlmSeverityError;
		tyAlmData.udiRunTime	:= tyAlmData.udiRunTime + 1;
		tyAlmData.bAlm			:= TRUE;
		tyAlmData.udiModuleNum  := udiModuleNum;
		g_sMachineProgNm		:= p_sProgNm;

		//Get Error Message
		IF tyAlmData.udiCode < 10000 OR tyAlmData.udiCode > 10099 THEN
			tyAlmData.sAlmMsg	:= 'Unknown';
			tyAlmData.sRcyMsg	:= 'Unknown';
		ELSE
			tyAlmData.sAlmMsg	:= a_tyAlmText[tyAlmData.udiCode].sAlmText;
			tyAlmData.sRcyMsg	:= a_tyAlmText[tyAlmData.udiCode].sRcyText;
		END_IF

	END_IF

END_ACTION
```

#### Act_AlarmInfo1.st - Change By Project
```iecst
(** 2019-03-25 **)
ACTION Act_Alarm1:

	//Error
	IF EDGEPOS(eStatus1 = Error) THEN

		tyAlmData1.sProgNm		:= p_sProgNm;
		tyAlmData1.udiCode		:= udiStatus1;
		tyAlmData1.eSeverity	:= AlmSeverityError;
		tyAlmData1.udiRunTime	:= tyAlmData1.udiRunTime + 1;
		tyAlmData1.bAlm			:= TRUE;
		tyAlmData1.udiModuleNum  := udiModuleNum;
		g_sMachineProgNm		:= p_sProgNm;

		//Get Error Message
		IF tyAlmData1.udiCode < 10000 OR tyAlmData1.udiCode > 10099 THEN
			tyAlmData1.sAlmMsg	:= 'Unknown';
			tyAlmData1.sRcyMsg	:= 'Unknown';
		ELSE
			tyAlmData1.sAlmMsg	:= a_tyAlmText[tyAlmData1.udiCode].sAlmText;
			tyAlmData1.sRcyMsg	:= a_tyAlmText[tyAlmData1.udiCode].sRcyText;
		END_IF

	END_IF

END_ACTION
```

#### InputRef.var - Change By Project
```iecst
(*2020-10-06*)
(**)
(*General*)
VAR
	p_udiRstErr : REFERENCE TO UDINT;
END_VAR
(**)
(*Configuration*)
VAR
	p_tyNtParamCurr : REFERENCE TO tyNtParam;
	p_bOpsRun : REFERENCE TO BOOL;
	p_bDIThermalPrtSig : REFERENCE TO BOOL;
	p_bDIPressureSW : REFERENCE TO BOOL;
END_VAR
(**)
(*Input*)
VAR
	p_sProgNm : REFERENCE TO STRING[15];
	p_bNtSettingsLoadDone : REFERENCE TO BOOL;
END_VAR
```

#### Local.var - Change By Project
```iecst
(*2020-10-06*)
(**)
(*Local Action, State & Status*)
VAR
	eStatus : eFBStatus := Idle;
	eStatus1 : eFBStatus := Idle;
	udiStatus : UDINT := 0;
	udiStatus1 : UDINT := 0;
END_VAR
(**)
(*Local Alarm*)
VAR
	tyAlmData : tyAlmDat;
	tyAlmData1 : tyAlmDat;
	a_tyAlmText : ARRAY[10000..10099] OF tyAlmTxt := [(sAlmText:='Pressure Switch Not Activated.',sRcyText:='Open Pneumatic Valve / Supply Air To Air Regulator.'),(sAlmText:='Thermal Protection Signal Not Activated.',sRcyText:='Check Signal and Part.'),98(0)];
END_VAR
(**)
(*Local Output*)
(**)
(*Local Input*)
VAR
	udiRstErr : UDINT := 0;
END_VAR
(**)
VAR
	sProgNm : STRING[15] := 'Machine';
	bNtSettingsLoadDone : BOOL := TRUE;
END_VAR
(**)
(*Local*)
VAR
	tyNtParamCurr : tyNtParam;
	bPressureSW : BOOL;
	bThermalPrtSig : BOOL;
	bRstErr : BOOL;
	udiRstErrOld : UDINT;
	bInitDone : BOOL;
	bInitialDone : BOOL;
	udiModuleNum : UDINT := 5951;
END_VAR
```

### MotorBrk.typ - Do Not Change!!!
```iecst
(*2018-12-14*)
(**)
(*Action*)

TYPE
	eMotorBrkAction :
		(
		MotorBrkActIdle,
		MotorBrkActCW,
		MotorBrkActCCW,
		MotorBrkActCCWSenToMidSen,
		MotorBrkActMidSenToCWSen,
		MotorBrkActCWSenToMidSen,
		MotorBrkActMidSenToCCWSen,
		MotorBrkActBrkRlsOn,
		MotorBrkActBrkRlsOff,
		MotorBrkActStop,
		MotorBrkActSetMtrSigOnOrCW,
		MotorBrkActSetMtrDirOrCCW,
		MotorBrkActSetMtrBrkRls,
		MotorBrkActRstMtrSigOnOrCW,
		MotorBrkActRstMtrDirOrCCW,
		MotorBrkActRstMtrBrkRls,
		MotorBrkActSetMtrAll,
		MotorBrkActRstMtrAll,
		MotorBrkActSetMtrDirOrCCW1,
		MotorBrkActRstMtrDirOrCCW1
		);
END_TYPE
```

### MotorBrk.var - Change By Project
```iecst
(*2019-03-25*)
(**)
(*Action & State & Status*)
VAR
	p_MotorBrkStat : UDINT;
	p_MotorBrkStatus : UDINT;
	p_MotorBrkStatTxt : UDINT;
END_VAR
(**)
(*Alarm*)
VAR
	p_MotorBrkAlmData : UDINT;
END_VAR
(**)
(*Output*)
VAR
	p_MotorBrkMtrSigOnOrCW : UDINT;
	p_MotorBrkMtrDirOrCCW : UDINT;
	p_MotorBrkMtrBrkRls : UDINT;
END_VAR
```

### Program Logical/MotorBrk/MotorBrk (IEC, version 1.00.0) - 1.00.0 - NtConv v5.00.0

#### Init.st - Change By Project
```iecst
(** 2019-03-25 **)
PROGRAM _INIT

	(* Always Change If Project Change *)

	//Pass Address To Global Address For External Use
	//Action, State & Status
	p_MotorBrkStat		:= ADR(eStat);
	p_MotorBrkStatus	:= ADR(eStatus);
	p_MotorBrkStatTxt	:= ADR(sStatTxt);

	//Alarm
	p_MotorBrkAlmData	:= ADR(tyAlmData);

	//Output
	p_MotorBrkMtrSigOnOrCW	:= ADR(bMtrSigOnOrCW);
	p_MotorBrkMtrDirOrCCW	:= ADR(bMtrDirOrCCW);
	p_MotorBrkMtrBrkRls		:= ADR(bMtrBrkRls);

	(* Always Change If Project Change *)

END_PROGRAM
```

#### Act_InitGlobal.st - Change By Project
```iecst
(** 2020-10-14 **)
ACTION Act_InitGlobal:

	(* Always Change If Project Change *)

	//Pass Data To Link
	p_bLinkOpsRun ACCESS p_OpsRun;
	p_bLinkOpsSimu ACCESS p_SimuRun;

	//Pass Data To Internal Use
	p_udiRstErr ACCESS p_RstErrReset;
	p_bManual ACCESS p_UIMnlMod;
	p_bNtSettingsLoadDone ACCESS p_StartupNtSettingsLoadDone;

	p_bCWSen ACCESS p_DIInvertRemoteSen;
	p_bCCWSen ACCESS p_DIInvertHomeSen;

	p_diMtrOnDlyTm ACCESS p_NtParamMotorOnDlyTm;
	p_diMtrOffDlyTm ACCESS p_NtParamMotorOffDlyTm;
	p_diBrkOnDlyTm ACCESS p_NtParamBrakeOnDlyTm;
	p_diBrkOffDlyTm ACCESS p_NtParamBrakeOffDlyTm;
	p_diTimeOut ACCESS p_NtParamTimeOut;

	p_bInletShutterCloseRS ACCESS p_DIInShutterCloseRS;
	p_bOutletShutterCloseRS ACCESS p_DIOutShutterCloseRS;
	p_bInletShutterPrep ACCESS p_NtParamProjInletShutPrep;
	p_bInletShutterDis ACCESS p_McParamInShutterDis;
	p_bOutletShutterPrep ACCESS p_NtParamProjOutletShutPrep;
	p_bOutletShutterDis ACCESS p_McParamOutShutterDis;

	(* Always Change If Project Change *)

END_ACTION
```

#### InputRef_Link.var - Change By Project
```iecst
(*2019-04-09*)
(**)
VAR
	p_bLinkOpsRun : REFERENCE TO BOOL;
	p_bLinkOpsSimu : REFERENCE TO BOOL;
END_VAR
```

#### Act_LinkAction.st - Change By Project
```iecst
(** 2019-04-09 **)
ACTION Act_LinkAction:

	IF p_bLinkOpsRun = TRUE THEN
		p_eAct ACCESS p_OpsInvertInvertAct;
	ELSIF p_bLinkOpsSimu THEN
		p_eAct ACCESS p_SimuInvInvAct;
	ELSIF p_bManual = TRUE THEN
		p_eAct ACCESS p_UIInvertAct;
	ELSE
		p_eAct ACCESS ADR(eAct);
	END_IF

END_ACTION
```

#### Act_Link.st - Change By Project
```iecst
(** 2020-10-14 **)
ACTION Act_Link:

	IF (p_bInletShutterPrep AND p_bInletShutterDis=FALSE) AND (p_bOutletShutterPrep AND p_bOutletShutterDis=FALSE) THEN
		p_bInterruptSensor := (p_bInletShutterCloseRS=FALSE) OR (p_bOutletShutterCloseRS=FALSE);

	ELSIF (p_bInletShutterPrep AND p_bInletShutterDis=FALSE) THEN
		p_bInterruptSensor := (p_bInletShutterCloseRS=FALSE);

	ELSIF (p_bInletShutterPrep AND p_bInletShutterDis=FALSE) THEN
		p_bInterruptSensor := (p_bOutletShutterCloseRS=FALSE);

	ELSE
		p_bInterruptSensor := FALSE;
	END_IF

END_ACTION
```

#### Cyclic.st - Do Not Change!!!
```iecst
(** 2019-03-29 **)
PROGRAM _CYCLIC

	IF bInitDone = FALSE THEN
		bInitDone	:= TRUE;

		Act_InitLocal;
		Act_InitGlobal;

	ELSIF bInitialDone = FALSE THEN
		IF p_bNtSettingsLoadDone = TRUE THEN
			bInitialDone	:= TRUE;

			Act_Initial;
		END_IF

	ELSE

		Act_RstErr;
		Act_LinkAction;
		Act_Action;
		Act_LinkEn;

		IF (p_bPrep = TRUE) AND (p_bEn = TRUE) AND (p_bDis = FALSE) THEN
			Act_Link;
			Act_Main;
			Act_Background;
		ELSE
			IF eStat <> MotorBrkActIdle THEN
				eStatus	:= Done;
			ELSE
				eStatus	:= Idle;
			END_IF
		END_IF

		Act_Alarm;

	END_IF

END_PROGRAM
```

#### Act_InitLocal.st - Do Not Change!!!
```iecst
(** 2020-10-14 **)
ACTION Act_InitLocal:

	//Input Reference Link To Local Variable
	p_eAct ACCESS ADR(eAct);
	p_udiRstErr ACCESS ADR(udiRstErr);
	p_bPrep ACCESS ADR(bPrep);
	p_bEn ACCESS ADR(bEn);
	p_bDis ACCESS ADR(bDis);
	p_bManual ACCESS ADR(bManual);
	p_bOnDirMod ACCESS ADR(bOnDirMod);
	p_diMtrSigOnDlyTm ACCESS ADR(diMtrSigOnDlyTm); //For Signal On Delay between Dir Rly and Run Rly
	p_diMtrDirOffDlyTm ACCESS ADR(diMtrDirOffDlyTm); //For Signal Off Delay between Run Rly and Dir Rly
	p_diMtrBrkOnDlyTm ACCESS ADR(diMtrBrkOnDlyTm); //For Signal Brake On Delay Tm
	p_diMtrOnDlyTm ACCESS ADR(diMtrOnDlyTm);
	p_diMtrOffDlyTm ACCESS ADR(diMtrOffDlyTm);
	p_diBrkOnDlyTm ACCESS ADR(diBrkOnDlyTm);
	p_diBrkOffDlyTm ACCESS ADR(diBrkOffDlyTm);
	p_diTimeOut ACCESS ADR(diTimeOut);
	p_sProgNm ACCESS ADR(sProgNm);
	p_bNtSettingsLoadDone ACCESS ADR(bNtSettingsLoadDone);
	p_bCCWSen ACCESS ADR(bCCWSen);
	p_bMidSen ACCESS ADR(bMidSen);
	p_bCWSen ACCESS ADR(bCWSen);
	p_bInterruptSensor ACCESS ADR(bInterruptSensor);

	p_bInletShutterCloseRS ACCESS ADR(bInletShutterCloseRS);
	p_bOutletShutterCloseRS ACCESS ADR(bOutletShutterCloseRS);
	p_bInletShutterPrep ACCESS ADR(bInletShutterPrep);
	p_bInletShutterDis ACCESS ADR(bInletShutterDis);
	p_bOutletShutterPrep ACCESS ADR(bOutletShutterPrep);
	p_bOutletShutterDis ACCESS ADR(bOutletShutterDis);

END_ACTION
```

#### Act_Initial.st - Do Not Change!!!
```iecst
(** 2019-03-22 **)
ACTION Act_Initial:

	//Initial
	sStatTxt	:= a_sStatText[eStat];

	fbRotCW.bOnDirMod		:= p_bOnDirMod;
	fbRotCW.tMtrOnDlyTm		:= DINT_TO_TIME(p_diMtrOnDlyTm);
	fbRotCW.tMtrOffDlyTm	:= DINT_TO_TIME(p_diMtrOffDlyTm);
	fbRotCW.tBrkOnDlyTm		:= DINT_TO_TIME(p_diBrkOnDlyTm);
	fbRotCW.tBrkOffDlyTm	:= DINT_TO_TIME(p_diBrkOffDlyTm);
	fbRotCW.tTxDlyTm		:= DINT_TO_TIME(p_diTimeOut);
	fbRotCW.tMtrSigOnDlyTm		:= DINT_TO_TIME(p_diMtrSigOnDlyTm);			//Locally
	fbRotCW.tMtrDirOffDlyTm		:= DINT_TO_TIME(p_diMtrDirOffDlyTm);		//Locally
//	fbRotCW.tMtrBrkOnDlyTm		:= DINT_TO_TIME(p_diMtrBrkOnDlyTm);			//Locally
	fbRotCW.bStartSen		:= TRUE;
	fbRotCW.bConvLToR		:= TRUE;
	fbRotCW(bEn := FALSE);

	fbRotCCW.bOnDirMod		:= p_bOnDirMod;
	fbRotCCW.tMtrOnDlyTm	:= DINT_TO_TIME(p_diMtrOnDlyTm);
	fbRotCCW.tMtrOffDlyTm	:= DINT_TO_TIME(p_diMtrOffDlyTm);
	fbRotCCW.tBrkOnDlyTm	:= DINT_TO_TIME(p_diBrkOnDlyTm);
	fbRotCCW.tBrkOffDlyTm	:= DINT_TO_TIME(p_diBrkOffDlyTm);
	fbRotCCW.tTxDlyTm		:= DINT_TO_TIME(p_diTimeOut);
	fbRotCCW.bStartSen		:= TRUE;
	fbRotCCW.bConvLToR		:= FALSE;
	fbRotCCW(bEn := FALSE);

	fbMtrBrkRlsOn(bEn := FALSE);
	fbMtrBrkRlsOff(bEn := FALSE);

	fbStop(bEn := FALSE);

END_ACTION
```

#### Act_Action.st - Do Not Change!!!
```iecst
(** 2020-10-14 **)
ACTION Act_Action:

	//Reset Error
	IF (eStatus = Error) AND bRstErr THEN
		p_eAct	:= MotorBrkActIdle;
		eStat	:= MotorBrkActIdle;
	END_IF

	//Set p_eAct
	IF eStatus = Idle OR eStatus = Busy OR eStatus = Done THEN
		eStat	:= p_eAct;
	END_IF

END_ACTION
```

#### Act_Main.st - Do Not Change!!!
```iecst
(** 2019-03-22 **)
ACTION Act_Main:

	IF eStatOld <> eStat THEN
		fbRotCW(bEn := FALSE);
		fbRotCCW(bEn := FALSE);
		fbStop(bEn := FALSE);
		fbMtrBrkRlsOn(bEn := FALSE);
		fbMtrBrkRlsOff(bEn := FALSE);
		fbMtrSigOnDlyTm(IN := FALSE);
		fbMtrDirOffDlyTm(IN := FALSE);

		IF eStatOld <> MotorBrkActIdle
			AND eStatOld <> MotorBrkActSetMtrSigOnOrCW
			AND eStatOld <> MotorBrkActSetMtrDirOrCCW
			AND eStatOld <> MotorBrkActSetMtrBrkRls
			AND eStatOld <> MotorBrkActRstMtrSigOnOrCW
			AND eStatOld <> MotorBrkActRstMtrDirOrCCW
			AND eStatOld <> MotorBrkActRstMtrBrkRls
			AND eStatOld <> MotorBrkActSetMtrAll
			AND eStatOld <> MotorBrkActRstMtrAll
			AND eStatOld <> MotorBrkActSetMtrDirOrCCW1
			AND eStatOld <> MotorBrkActRstMtrDirOrCCW1
			THEN

			bMtrSigOnOrCW	:= FALSE;
			bMtrDirOrCCW	:= FALSE;
			bMtrBrkRls		:= FALSE;

		END_IF

		sStatTxt	:= a_sStatText[eStat];

		eStatOld	:= eStat;

		eStatus		:= Busy;
	END_IF

	//Main
	CASE eStat OF

		MotorBrkActIdle:
			IF EDGENEG(p_bManual) THEN
				bMtrSigOnOrCW	:= FALSE;
				bMtrDirOrCCW	:= FALSE;
				bMtrBrkRls		:= FALSE;
			END_IF

			eStatus	:= Idle;
			bNotInterruptible := FALSE ;

		MotorBrkActCW:

			IF eStatus = Idle OR eStatus = Busy THEN

				eStatus	:= Busy;

				bNotInterruptible := TRUE;

				//Motor Run
				fbRotCW.bEndSen			:= p_bCWSen;
				fbRotCW.bLmtSen			:= FALSE;

				fbRotCW(bEn := TRUE);

				bMtrSigOnOrCW	:= fbRotCW.bMtrSigOnOrLToR;
				bMtrDirOrCCW	:= fbRotCW.bMtrDirOrRToL;
				bMtrBrkRls		:= fbRotCW.bMtrBrk;

				IF fbRotCW.udiStatus = 0 THEN
					IF fbRotCW.bEndSen = TRUE THEN
						eStatus		:= Done;
					ELSE
						udiStatus	:= 10000;	//Motor Time Out While Turning Clockwise
						eStatus		:= Error;
					END_IF
				ELSIF fbRotCW.udiStatus < 65534 THEN
					udiStatus	:= fbRotCW.udiStatus;
					eStatus		:= Error;
				END_IF
			END_IF

		MotorBrkActCCW:

			IF eStatus = Idle OR eStatus = Busy THEN

				eStatus	:= Busy;

				bNotInterruptible := TRUE;

				//Motor Run
				fbRotCCW.bEndSen		:= p_bCCWSen;
				fbRotCCW.bLmtSen		:= FALSE;

				fbRotCCW(bEn := TRUE);

				bMtrSigOnOrCW	:= fbRotCCW.bMtrSigOnOrLToR;
				bMtrDirOrCCW	:= fbRotCCW.bMtrDirOrRToL;
				bMtrBrkRls		:= fbRotCCW.bMtrBrk;

				IF fbRotCCW.udiStatus = 0 THEN
					IF fbRotCCW.bEndSen = TRUE THEN
						eStatus		:= Done;
					ELSE
						udiStatus	:= 10001;	//Motor Time Out While Turning Counter Clockwise
						eStatus		:= Error;
					END_IF
				ELSIF fbRotCCW.udiStatus < 65534 THEN
					udiStatus	:= fbRotCCW.udiStatus;
					eStatus		:= Error;
				END_IF
			END_IF

		MotorBrkActCCWSenToMidSen:
			bNotInterruptible := TRUE;
			IF eStatus = Idle OR eStatus = Busy THEN

				eStatus	:= Busy;

				bNotInterruptible := TRUE;

				//Motor Run
				fbRotCW.bEndSen			:= p_bMidSen;
				fbRotCW.bLmtSen			:= p_bCWSen;

				fbRotCW(bEn := TRUE);

				bMtrSigOnOrCW	:= fbRotCW.bMtrSigOnOrLToR;
				bMtrDirOrCCW	:= fbRotCW.bMtrDirOrRToL;
				bMtrBrkRls		:= fbRotCW.bMtrBrk;

				IF fbRotCW.udiStatus = 0 THEN
					IF fbRotCW.bLmtActivated = TRUE THEN
						udiStatus	:= 10002;	//Clockwise Sensor Activated While Turning Clockwise To Middle Sensor
						eStatus		:= Error;
					ELSIF fbRotCW.bEndSen = TRUE THEN
						eStatus		:= Done;
					ELSE
						udiStatus	:= 10003;	//Motor Time Out While Turning Clockwise To Middle Sensor
						eStatus		:= Error;
					END_IF
				ELSIF fbRotCW.udiStatus < 65534 THEN
					udiStatus	:= fbRotCW.udiStatus;
					eStatus		:= Error;
				END_IF
			END_IF

		MotorBrkActMidSenToCWSen:

			IF eStatus = Idle OR eStatus = Busy THEN

				eStatus	:= Busy;

				bNotInterruptible := TRUE;

				//Motor Run
				fbRotCW.bEndSen			:= p_bCWSen;
				fbRotCW.bLmtSen			:= FALSE;

				fbRotCW(bEn := TRUE);

				bMtrSigOnOrCW	:= fbRotCW.bMtrSigOnOrLToR;
				bMtrDirOrCCW	:= fbRotCW.bMtrDirOrRToL;
				bMtrBrkRls		:= fbRotCW.bMtrBrk;

				IF fbRotCW.udiStatus = 0 THEN
					IF fbRotCW.bEndSen = TRUE THEN
						eStatus		:= Done;
					ELSE
						udiStatus	:= 10004;	//Motor Time Out While Turning Clockwise From Middle Sensor
						eStatus		:= Error;
					END_IF
				ELSIF fbRotCW.udiStatus < 65534 THEN
					udiStatus	:= fbRotCW.udiStatus;
					eStatus		:= Error;
				END_IF
			END_IF

		MotorBrkActCWSenToMidSen:

			IF eStatus = Idle OR eStatus = Busy THEN

				eStatus	:= Busy;

				bNotInterruptible := TRUE;

				//Motor Run
				fbRotCCW.bEndSen		:= p_bMidSen;
				fbRotCCW.bLmtSen		:= p_bCCWSen;

				fbRotCCW(bEn := TRUE);

				bMtrSigOnOrCW	:= fbRotCCW.bMtrSigOnOrLToR;
				bMtrDirOrCCW	:= fbRotCCW.bMtrDirOrRToL;
				bMtrBrkRls		:= fbRotCCW.bMtrBrk;

				IF fbRotCCW.udiStatus = 0 THEN
					IF fbRotCCW.bLmtActivated = TRUE THEN
						udiStatus	:= 10005;	//Counter Clockwise Sensor Activated While Turning Counter Clockwise To Middle Sensor
						eStatus		:= Error;
					ELSIF fbRotCCW.bEndSen = TRUE THEN
						eStatus		:= Done;
					ELSE
						udiStatus	:= 10006;	//Motor Time Out While Turning Counter Clockwise To Middle Sensor
						eStatus		:= Error;
					END_IF
				ELSIF fbRotCCW.udiStatus < 65534 THEN
					udiStatus	:= fbRotCCW.udiStatus;
					eStatus		:= Error;
				END_IF
			END_IF

		MotorBrkActMidSenToCCWSen:

			IF eStatus = Idle OR eStatus = Busy THEN

				eStatus	:= Busy;

				bNotInterruptible := TRUE;

				//Motor Run
				fbRotCCW.bEndSen		:= p_bCCWSen;
				fbRotCCW.bLmtSen		:= FALSE;

				fbRotCCW(bEn := TRUE);

				bMtrSigOnOrCW	:= fbRotCCW.bMtrSigOnOrLToR;
				bMtrDirOrCCW	:= fbRotCCW.bMtrDirOrRToL;
				bMtrBrkRls		:= fbRotCCW.bMtrBrk;

				IF fbRotCCW.udiStatus = 0 THEN
					IF fbRotCCW.bEndSen = TRUE THEN
						eStatus		:= Done;
					ELSE
						udiStatus	:= 10007;	//Motor Time Out While Turning Counter Clockwise From Middle Sensor
						eStatus		:= Error;
					END_IF
				ELSIF fbRotCCW.udiStatus < 65534 THEN
					udiStatus	:= fbRotCCW.udiStatus;
					eStatus		:= Error;
				END_IF
			END_IF

		MotorBrkActBrkRlsOn:

			IF eStatus = Idle OR eStatus = Busy THEN

				eStatus	:= Busy;

				//Motor Run
				fbMtrBrkRlsOn(bEn := TRUE);

				bMtrBrkRls	:= fbMtrBrkRlsOn.bMtrBrk;

				IF fbMtrBrkRlsOn.udiStatus = 0 THEN
					eStatus		:= Done;
				ELSIF fbMtrBrkRlsOn.udiStatus < 65534 THEN
					udiStatus	:= fbMtrBrkRlsOn.udiStatus;
					eStatus		:= Error;
				END_IF
			END_IF

		MotorBrkActBrkRlsOff:
			IF eStatus = Idle OR eStatus = Busy THEN

				eStatus	:= Busy;

				//Motor Run
				fbMtrBrkRlsOff(bEn := TRUE);

				bMtrBrkRls	:= fbMtrBrkRlsOff.bMtrBrk;

				IF fbMtrBrkRlsOff.udiStatus = 0 THEN
					eStatus		:= Done;
				ELSIF fbMtrBrkRlsOff.udiStatus < 65534 THEN
					udiStatus	:= fbMtrBrkRlsOff.udiStatus;
					eStatus		:= Error;
				END_IF
			END_IF

		MotorBrkActStop:
			IF eStatus = Idle OR eStatus = Busy THEN

				eStatus	:= Busy;

				//Motor Run
				fbStop(bEn := TRUE);
				fbMtrBrkRlsOff(bEn := TRUE);

				bMtrSigOnOrCW	:= fbStop.bMtrSigOnOrLToR;
				bMtrDirOrCCW	:= fbStop.bMtrDirOrRToL;
				bMtrBrkRls		:= fbMtrBrkRlsOff.bMtrBrk;

				IF fbStop.udiStatus = 0 AND fbMtrBrkRlsOff.udiStatus = 0 THEN
					eStatus	:= Done;
				ELSIF fbStop.udiStatus < 65534 AND fbStop.udiStatus > 0 THEN
					udiStatus	:= fbStop.udiStatus;
					eStatus		:= Error;
				ELSIF fbMtrBrkRlsOff.udiStatus < 65534 AND fbMtrBrkRlsOff.udiStatus > 0 THEN
					udiStatus	:= fbMtrBrkRlsOff.udiStatus;
					eStatus		:= Error;
				END_IF
			END_IF

		MotorBrkActSetMtrSigOnOrCW:

			IF eStatus = Idle OR eStatus = Busy THEN

				bNotInterruptible := TRUE;

				bMtrSigOnOrCW	:= TRUE;
				eStatus			:= Done;

			END_IF

		MotorBrkActSetMtrDirOrCCW:

			IF eStatus = Idle OR eStatus = Busy THEN

				bNotInterruptible := TRUE;

				bMtrDirOrCCW	:= TRUE;
				eStatus			:= Done;

			END_IF

		MotorBrkActSetMtrDirOrCCW1:

			IF eStatus = Idle OR eStatus = Busy THEN

				bNotInterruptible := TRUE;

				bMtrDirOrCCW	:= TRUE;
				fbMtrSigOnDlyTm (IN:= TRUE);

				IF fbMtrSigOnDlyTm.Q THEN
					bMtrSigOnOrCW	:= TRUE;
					fbMtrSigOnDlyTm (IN:= FALSE);
					eStatus			:= Done;
				END_IF
//				bMtrSigOnOrCW	:= TRUE;
//				bMtrDirOrCCW	:= TRUE;
//				eStatus			:= Done;
			END_IF

		MotorBrkActSetMtrBrkRls:
			IF eStatus = Idle OR eStatus = Busy THEN

				bMtrBrkRls		:= TRUE;
				eStatus			:= Done;

			END_IF

		MotorBrkActRstMtrSigOnOrCW:
			IF eStatus = Idle OR eStatus = Busy THEN

				bMtrSigOnOrCW	:= FALSE;
				eStatus			:= Done;

			END_IF

		MotorBrkActRstMtrDirOrCCW:

			IF eStatus = Idle OR eStatus = Busy THEN

				bMtrDirOrCCW	:= FALSE;
				eStatus			:= Done;

			END_IF

		MotorBrkActRstMtrDirOrCCW1:
			IF eStatus = Idle OR eStatus = Busy THEN

				fbMtrDirOffDlyTm (IN:=TRUE);
				IF 	fbMtrDirOffDlyTm.Q THEN
					fbMtrDirOffDlyTm (IN:=FALSE);
					bMtrDirOrCCW	:= FALSE;
					eStatus			:= Done;
				END_IF
				bMtrSigOnOrCW	:= FALSE;

			END_IF

		MotorBrkActRstMtrBrkRls:
			IF eStatus = Idle OR eStatus = Busy THEN

				bMtrBrkRls		:= FALSE;
				eStatus			:= Done;

			END_IF

		MotorBrkActSetMtrAll:

			IF eStatus = Idle OR eStatus = Busy THEN

				bNotInterruptible := TRUE;

				bMtrSigOnOrCW	:= TRUE;
				bMtrDirOrCCW	:= TRUE;
				bMtrBrkRls		:= TRUE;
				eStatus			:= Done;

			END_IF

		MotorBrkActRstMtrAll:
			IF eStatus = Idle OR eStatus = Busy THEN

				bMtrSigOnOrCW	:= FALSE;
				bMtrDirOrCCW	:= FALSE;
				bMtrBrkRls		:= FALSE;
				eStatus			:= Done;

			END_IF

	END_CASE

END_ACTION
```

#### Act_Background.st - Do Not Change!!!
```iecst
(** 2020-10-14 **)
ACTION Act_Background:

	IF bNotInterruptible THEN
		IF p_bInterruptSensor = TRUE THEN
			eStatus	:= Error;
			udiStatus	:= 10008;	//Sensor Interrupt Motor Movement

			p_eAct	:= MotorBrkActIdle;
			eStat	:= MotorBrkActIdle;
		END_IF
	END_IF

END_ACTION
```

#### Act_Alarm.st - Do Not Change!!!
```iecst
(** 2019-03-25 **)
ACTION Act_Alarm:

	//Error
	IF EDGEPOS(eStatus = Error) THEN

		tyAlmData.sProgNm		:= p_sProgNm;
		tyAlmData.udiCode		:= udiStatus;
		tyAlmData.eSeverity		:= AlmSeverityError;
		tyAlmData.udiRunTime	:= tyAlmData.udiRunTime + 1;
		tyAlmData.bAlm			:= TRUE;
		tyAlmData.udiModuleNum  := udiModuleNum;
		g_sMotorBrkProgNm		:= p_sProgNm;

		//Get Error Message
		IF tyAlmData.udiCode < 10000 OR tyAlmData.udiCode > 10099 THEN
			tyAlmData.sAlmMsg	:= 'Unknown';
			tyAlmData.sRcyMsg	:= 'Unknown';
		ELSE
			tyAlmData.sAlmMsg	:= a_tyAlmText[tyAlmData.udiCode].sAlmText;
			tyAlmData.sRcyMsg	:= a_tyAlmText[tyAlmData.udiCode].sRcyText;
		END_IF

		sStatTxt	:= tyAlmData.sAlmMsg;

	ELSIF bRstErr AND (tyAlmData.udiCode <> 0) THEN

		tyAlmData.udiCode	:= 0;
		tyAlmData.eSeverity	:= AlmSeverityNA;
		tyAlmData.sAlmMsg	:= '';
		tyAlmData.sRcyMsg	:= '';
		tyAlmData.bAlm		:= FALSE;
		sStatTxt	:= a_sStatText[eStat];

	END_IF

END_ACTION
```

#### InputRef.var - Do Not Change!!!
```iecst
(*2020-10-14*)
(**)
(*General*)
VAR
	p_eAct : REFERENCE TO eMotorBrkAction;
	p_udiRstErr : REFERENCE TO UDINT;
	p_bPrep : REFERENCE TO BOOL;
	p_bEn : REFERENCE TO BOOL;
	p_bDis : REFERENCE TO BOOL;
END_VAR
(**)
(*Configuration*)
VAR
	p_bManual : REFERENCE TO BOOL;
	p_bOnDirMod : REFERENCE TO BOOL;
	p_diMtrSigOnDlyTm : REFERENCE TO DINT;
	p_diMtrDirOffDlyTm : REFERENCE TO DINT;
	p_diMtrBrkOnDlyTm : REFERENCE TO DINT;
	p_diMtrOnDlyTm : REFERENCE TO DINT;
	p_diMtrOffDlyTm : REFERENCE TO DINT;
	p_diBrkOnDlyTm : REFERENCE TO DINT;
	p_diBrkOffDlyTm : REFERENCE TO DINT;
	p_diTimeOut : REFERENCE TO DINT;
	p_sProgNm : REFERENCE TO STRING[15];
	p_bNtSettingsLoadDone : REFERENCE TO BOOL;
	p_bInletShutterCloseRS : REFERENCE TO BOOL;
	p_bOutletShutterCloseRS : REFERENCE TO BOOL;
	p_bInletShutterPrep : REFERENCE TO BOOL;
	p_bInletShutterDis : REFERENCE TO BOOL;
	p_bOutletShutterPrep : REFERENCE TO BOOL;
	p_bOutletShutterDis : REFERENCE TO BOOL;
END_VAR
(**)
(*Input*)
VAR
	p_bCCWSen : REFERENCE TO BOOL;
	p_bMidSen : REFERENCE TO BOOL;
	p_bCWSen : REFERENCE TO BOOL;
	p_bLiftRemoteSen : REFERENCE TO BOOL;
	p_bLiftHomeSen : REFERENCE TO BOOL;
	p_bSensor1 : REFERENCE TO BOOL;
	p_bSensor2 : REFERENCE TO BOOL;
	p_bSensor3 : REFERENCE TO BOOL;
	p_bInterruptSensor : REFERENCE TO BOOL;
	p_rMcParamStepper180deg : REFERENCE TO REAL;
	p_rMcParamStepperNeg90deg : REFERENCE TO REAL;
	p_rMcParamStepper90deg : REFERENCE TO REAL;
	p_rMcParamStepper0deg : REFERENCE TO REAL;
END_VAR
```

#### Local.var - Do Not Change!!!
```iecst
(*2019-04-30*)
(**)
(*Local Action, State & Status*)
VAR
	eAct : eMotorBrkAction := MotorBrkActIdle;
	eStat : eMotorBrkAction := MotorBrkActIdle;
	eStatus : eFBStatus := Idle;
	udiStatus : UDINT := 0;
	sStatTxt : STRING[200] := '';
	a_sStatText : ARRAY[0..50] OF STRING[200] := ['Idling','Turning Clockwise','Turning Counter Clockwise','Turning Clockwise From CCW Sensor To Middle Sensor','Turning Clockwise From Middle Sensor To CW Sensor','Turning Counter Clockwise From CW Sensor To Middle Sensor','Turning Counter Clockwise From Middle Sensor To CCW Sensor','Powering On Break Release','Powering Off Break Release','Stopping','Turning On Motor Signal','Turning On Motor Direction','Turning On Motor Break Release','Turning Off Motor Signal','Turning Off Motor Direction','Turning Off Motor Break Release','Turning On All Motor Output','Turning Off All Motor Output',33('')];
END_VAR
(**)
(*Local Alarm*)
VAR
	tyAlmData : tyAlmDat;
	a_tyAlmText : ARRAY[10000..10099] OF tyAlmTxt := [(sAlmText:='Motor Time Out While Turning Clockwise',sRcyText:='Motor Timeout Expired Before Operation Completed. Motor Operation Is Abnormal. Solve The Error To Resume Operation.'),(sAlmText:='Motor Time Out While Turning Counter Clockwise',sRcyText:='Motor Timeout Expired Before Operation Completed. Motor Operation Is Abnormal. Solve The Error To Resume Operation.'),(sAlmText:='Clockwise Sensor Activated While Turning Clockwise To Middle Sensor',sRcyText:='Incorrect Sensor Activated While Turning. Solve The Error To Resume Operation.'),(sAlmText:='Motor Time Out While Turning Clockwise To Middle Sensor',sRcyText:='Motor Timeout Expired Before Operation Completed. Motor Operation Is Abnormal. Solve The Error To Resume Operation.'),(sAlmText:='Motor Time Out While Turning Clockwise From Middle Sensor',sRcyText:='Motor Timeout Expired Before Operation Completed. Motor Operation Is Abnormal. Solve The Error To Resume Operation.'),(sAlmText:='Counter Clockwise Sensor Activated While Turning Counter Clockwise To Middle Sensor',sRcyText:='Incorrect Sensor Activated While Turning. Solve The Error To Resume Operation.'),(sAlmText:='Motor Time Out While Turning Counter Clockwise To Middle Sensor',sRcyText:='Motor Timeout Expired Before Operation Completed. Motor Operation Is Abnormal. Solve The Error To Resume Operation.'),(sAlmText:='Motor Time Out While Turning Counter Clockwise From Middle Sensor',sRcyText:='Motor Timeout Expired Before Operation Completed. Motor Operation Is Abnormal. Solve The Error To Resume Operation.'),(sAlmText:='Sensor Interrupt Motor Movement',sRcyText:='Operation Stop Due To The Interruption Of Sensor While Motor Moving. Solve The Interruption To Resume Operation.'),91((0))];
END_VAR
(**)
(*Local Output*)
VAR
	bMtrSigOnOrCW : BOOL := FALSE;
	bMtrDirOrCCW : BOOL := FALSE;
	bMtrBrkRls : BOOL := FALSE;
END_VAR
(**)
(*Local Input*)
VAR
	udiRstErr : UDINT := 0;
	bPrep : BOOL := TRUE;
	bEn : BOOL := TRUE;
	bDis : BOOL := FALSE;
	bManual : BOOL := FALSE;
	bOnDirMod : BOOL := FALSE;
	diMtrSigOnDlyTm : DINT := 500; (*For Sig On Dly*)
	diMtrDirOffDlyTm : DINT := 500; (*For Dir Off Dly*)
	diMtrBrkOnDlyTm : DINT := 100; (*For Mtr Brk Dly On Tm*)
	diMtrOnDlyTm : DINT := 500;
	diMtrOffDlyTm : DINT := 1000;
	diBrkOnDlyTm : DINT := 0;
	diBrkOffDlyTm : DINT := 500;
	diTimeOut : DINT := 10000;
	sProgNm : STRING[15] := 'MotorBrk';
	bNtSettingsLoadDone : BOOL := TRUE;
	bCCWSen : BOOL := FALSE;
	bMidSen : BOOL := FALSE;
	bCWSen : BOOL := FALSE;
	bInletShutterCloseRS : BOOL;
	bOutletShutterCloseRS : BOOL;
	bInletShutterPrep : BOOL;
	bInletShutterDis : BOOL;
	bOutletShutterPrep : BOOL;
	bOutletShutterDis : BOOL;
END_VAR
(**)
(*Local*)
VAR
	bRstErr : BOOL;
	udiRstErrOld : UDINT;
	bInitDone : BOOL;
	eStatOld : eMotorBrkAction := MotorBrkActIdle;
	bInitialDone : BOOL;
	fbRotCW : fbConvSenToSenBrkTmLmt;
	fbRotCCW : fbConvSenToSenBrkTmLmt;
	fbStop : fbConvMtrOff;
	fbMtrBrkRlsOn : fbConvBrkOn;
	fbMtrBrkRlsOff : fbConvBrkOff;
	bReached : BOOL;
	fbMtrSigOnDlyTm : TON := (PT:=T#200ms); (*Direct Ctrl Dly Tm for Run Rly*)
	fbMtrDirOffDlyTm : TON := (PT:=T#200ms); (*Direct Ctrl Dly Tm For Dir Rly*)
	bNotInterruptible : BOOL;
	bInterruptSensor : BOOL;
	b0Angle : BOOL := FALSE;
	bNeg90Angle : BOOL := FALSE;
	b90Angle : BOOL := FALSE;
	b180Angle : BOOL := FALSE;
	udiModuleNum : UDINT := 2101;
END_VAR
```

### Simu.typ - Do Not Change!!!
```iecst
(*2019-01-20*)
(**)

TYPE
	eSimulationsAction :
		(
		SimulationsActIdle,
		SimulationsActStart,
		SimulationsActStop,
		SimulationsActStep,
		SimulationsActError
		);
END_TYPE

(**)

TYPE
	eSimulationsStatus :
		(
		SimulationsStatusRun,
		SimulationsStatusStop,
		SimulationsStatusCycleStopping,
		SimulationsStatusStep
		);
END_TYPE
```

### Simu.var - Change By Project
```iecst
(*2019-01-20*)
(**)
(*Action & State & Status*)
VAR
	p_SimuAct : UDINT;
	p_SimuStat : UDINT;
	p_SimuStatus : UDINT;
	p_SimuStatTxt : UDINT;
END_VAR
(**)
(*Alarm*)
(**)
(*Output*)
VAR
	p_SimuSimuStatus : UDINT;
	p_SimuStatusRun : UDINT;
	p_SimuStatusStop : UDINT;
	p_SimuStatusCycleStop : UDINT;
	p_SimuStatusStep : UDINT;
	p_SimuRun : UDINT;
	p_SimuStop : UDINT;
	p_SimuStep : UDINT;
END_VAR
```

### Program Logical/Simulation/Simu (IEC, version 1.00.0) - 1.00.0 - 

#### Init.st - Change By Project
```iecst
(** 2019-03-25 **)
PROGRAM _INIT

	(* Always Change If Project Change *)

	//Pass Address To Global Address For External Use
	//Action, State & Status
	p_SimuStat		:= ADR(eStat);
	p_SimuStatus	:= ADR(eStatus);
	p_SimuStatTxt	:= ADR(sStatTxt);

	//Alarm

	//Output
	p_SimuSimuStatus		:= ADR(eSimuStatus);
	p_SimuStatusRun			:= ADR(bStatusRun);
	p_SimuStatusStop		:= ADR(bStatusStop);
	p_SimuStatusCycleStop	:= ADR(bStatusCycleStop);
	p_SimuStatusStep		:= ADR(bStatusStep);

	p_SimuRun				:= ADR(bRun);
	p_SimuStop				:= ADR(bStop);
	p_SimuStep				:= ADR(bStep);

	(* Always Change If Project Change *)

END_PROGRAM
```

#### Act_InitGlobal.st - Change By Project
```iecst
(** 2019-03-22 **)
ACTION Act_InitGlobal:

	(* Always Change If Project Change *)

	//Pass Data To Link
	p_eUISimuAct ACCESS p_UISimuAct;

	//Pass Data To Internal Use
	p_bSimuInvPaused ACCESS p_SimuInvPaused;
	p_bNtSettingsLoadDone ACCESS p_StartupNtSettingsLoadDone;

	(* Always Change If Project Change *)

END_ACTION
```

#### InputRef_Link.var - Change By Project
```iecst
(*2019-01-20*)
(**)
VAR
	p_eUISimuAct : REFERENCE TO eSimulationsAction;
	p_bSimuInvPaused : REFERENCE TO BOOL;
END_VAR
```

#### Act_LinkAction.st - Change By Project
```iecst
(** 2019-03-29 **)
ACTION Act_LinkAction:

	//Operation Control
	IF p_eUISimuAct <> SimulationsActIdle THEN
		p_eAct ACCESS p_UISimuAct;

	ELSE
		p_eAct ACCESS p_UISimuAct;

	END_IF

END_ACTION
```

#### Act_Link.st - Change By Project
```iecst
(** 2019-01-20 **)
ACTION Act_Link:

END_ACTION
```

#### Act_InitLocal.st - Do Not Change!!!
```iecst
(** 2019-03-25 **)
ACTION Act_InitLocal:

	//Input Reference Link To Local Variable
	p_eAct ACCESS ADR(eAct);
	p_udiRstErr ACCESS ADR(udiRstErr);
	p_bPaused ACCESS ADR(bPaused);
	p_bNtSettingsLoadDone ACCESS ADR(bNtSettingsLoadDone);

END_ACTION
```

#### Act_Initial.st - Do Not Change!!!
```iecst
(** 2019-01-08 **)
ACTION Act_Initial:

	//Initial
	sStatTxt	:= a_sStatText[eStat];

END_ACTION
```

#### Act_Action.st - Do Not Change!!!
```iecst
(** 2019-03-25 **)
ACTION Act_Action:

	//Reset Error
	IF (eStatus = Error) AND bRstErr THEN
		p_eAct	:= SimulationsActIdle;
		eStat	:= SimulationsActIdle;
	END_IF

	//Set p_eAct
	IF eStatus = Idle OR eStatus = Busy OR eStatus = Done THEN
		eStat	:= p_eAct;
	END_IF

END_ACTION
```

#### Act_Main.st - Do Not Change!!!
```iecst
(** 2019-01-20 **)
ACTION Act_Main:

	IF eStatOld <> eStat THEN
		usiStep		:= 0;

		sStatTxt	:= a_sStatText[eStat];

		eStatOld	:= eStat;

		eStatus		:= Busy;
	END_IF

	//Main
	CASE eStat OF

		SimulationsActIdle:
			eStatus	:= Idle;

		SimulationsActStart:
			IF eStatus = Idle OR eStatus = Busy THEN

				eSimuStatus			:= SimulationsStatusRun;
				bStatusRun			:= TRUE;
				bStatusStop			:= FALSE;
				bStatusCycleStop	:= FALSE;
				bStatusStep			:= FALSE;

				bRun		:= TRUE;
				bStop		:= FALSE;
				bStep		:= FALSE;

				eStatus	:= Done;

			END_IF

		SimulationsActStop:
			IF eStatus = Idle OR eStatus = Busy THEN

				eStatus	:= Busy;

				eSimuStatus			:= SimulationsStatusCycleStopping;
				bStatusRun			:= FALSE;
				bStatusStop			:= FALSE;
				bStatusCycleStop	:= TRUE;

				bStop	:= TRUE;

				IF p_bPaused THEN

					bRun	:= FALSE;

					eSimuStatus			:= SimulationsStatusStop;
					bStatusRun			:= FALSE;
					bStatusStop			:= TRUE;
					bStatusCycleStop	:= FALSE;

					eStatus	:= Done;

				END_IF

			END_IF

		SimulationsActStep:
			IF eStatus = Idle OR eStatus = Busy THEN

				eStatus	:= Busy;

				eSimuStatus			:= SimulationsStatusStep;
				bStatusRun			:= FALSE;
				bStatusStop			:= FALSE;
				bStatusCycleStop	:= FALSE;

				bRun	:= TRUE;

				CASE usiStep OF

					0:
						bStep	:= FALSE;
						usiStep	:= 1;

					1:
						bStep	:= TRUE;

				END_CASE

				IF p_bPaused THEN
					eStatus	:= Done;
				END_IF

			END_IF

		SimulationsActError:
			IF eStatus = Idle OR eStatus = Busy THEN

				eSimuStatus			:= SimulationsStatusStop;
				bStatusRun			:= FALSE;
				bStatusStop			:= TRUE;
				bStatusCycleStop	:= FALSE;

				bRun		:= FALSE;
				bStop		:= FALSE;
				bStep		:= FALSE;

				eStatus	:= Done;

			END_IF

	END_CASE

END_ACTION
```

#### InputRef.var - Do Not Change!!!
```iecst
(*2019-03-25*)
(**)
(*General*)
VAR
	p_eAct : REFERENCE TO eSimulationsAction;
	p_udiRstErr : REFERENCE TO UDINT;
	p_bPaused : REFERENCE TO BOOL;
	p_bNtSettingsLoadDone : REFERENCE TO BOOL;
END_VAR
```

#### Local.var - Do Not Change!!!
```iecst
(*2019-03-22*)
(**)
(*Local Action, State & Status*)
VAR
	eAct : eSimulationsAction := SimulationsActIdle;
	eStat : eSimulationsAction := SimulationsActIdle;
	eStatus : eFBStatus := Idle;
	sStatTxt : STRING[100] := '';
	a_sStatText : ARRAY[0..50] OF STRING[100] := ['Idling','Starting Operations','Sequence Stopping Operations','Pause Operations In Step','Accepting New Data','Accepted New Data','Error Immediate Stop Operations',44('')];
END_VAR
(**)
(*Local Alarm*)
(**)
(*Local Output*)
VAR
	eSimuStatus : eSimulationsStatus := SimulationsStatusStop;
	bStatusRun : BOOL;
	bStatusStop : BOOL := TRUE;
	bStatusCycleStop : BOOL;
	bStatusStep : BOOL;
	bRun : BOOL;
	bStop : BOOL;
	bStep : BOOL;
END_VAR
(**)
(*Local Input*)
VAR
	udiRstErr : UDINT := 0;
	bPaused : BOOL;
	bNtSettingsLoadDone : BOOL := TRUE;
END_VAR
(**)
(*Local*)
VAR
	bRstErr : BOOL;
	udiRstErrOld : UDINT;
	bInitDone : BOOL;
	bInitialDone : BOOL;
	eStatOld : eSimulationsAction := SimulationsActIdle;
	usiStep : USINT;
END_VAR
```

### SimuInv.var - Change By Project
```iecst
(*2019-03-25*)
(**)
(*Action & State & Status*)
(**)
(*Alarm*)
(**)
(*Output*)
VAR
	p_SimuInvPaused : UDINT;
END_VAR
(**)
VAR
	p_SimuInvInvAct : UDINT;
	p_SimuInvStopperAct : UDINT;
	p_SimuInvInShutterAct : UDINT;
	p_SimuInvOutShutterAct : UDINT;
	p_SimuInvConvAct : UDINT;
END_VAR
```

### SimuInv.typ - Do Not Change!!!
```iecst
(*2023_07_24*)
(**)
(*Sequence*)

TYPE
	eSimuInvRunStep :
		(
		SimuInvStepNA,
		SimuInvStepChkCondition,
		SimuInvStepInvertHome,
		SimuInvStepInvertRemote,
		SimuInvStepConvToRightSen,
		SimuInvStepConvToLeftSen,
		SimuInvStepInitShutterCls,
		SimuInvStepInitStopperExt
		);
END_TYPE
```

### Program Logical/Simulation/SimuInv (IEC, version 1.00.0) - 1.00.0 - 

#### Init.st - Change By Project
```iecst
(** 2022-09-15 **)
PROGRAM _INIT

	(* Always Change If Project Change *)

	//Pass Address To Global Address For External Use
	//Action, State & Status

	//Alarm

	//Output
	p_SimuInvPaused				:= ADR(bPaused);

	p_SimuInvInvAct				:= ADR(eInverterAct);
	p_SimuInvConvAct			:= ADR(eConvAct);
	p_SimuInvInShutterAct		:= ADR(eInShutterAct);
	p_SimuInvOutShutterAct		:= ADR(eOutShutterAct);
	p_SimuInvStopperAct			:= ADR(eStopperAct);

	(* Always Change If Project Change *)

END_PROGRAM
```

#### Act_InitGlobal.st - Change By Project
```iecst
(** 2019-03-22 **)
ACTION Act_InitGlobal:

	(* Always Change If Project Change *)

	//Pass Data To Link

	//Pass Data To Internal Use
	p_udiRstErr ACCESS p_RstErrReset;
	p_bRun ACCESS p_SimuRun;
	p_bStop ACCESS p_SimuStop;
	p_bStep ACCESS p_SimuStep;
	p_bNtSettingsLoadDone ACCESS p_StartupNtSettingsLoadDone;
	p_bInletShutterPrep ACCESS p_NtParamProjInletShutPrep;
	p_bOutletShutterPrep ACCESS p_NtParamProjOutletShutPrep;

	p_eInvertStat ACCESS p_MotorBrkStat;
	p_eInvertStatus ACCESS p_MotorBrkStatus;
	p_bInverterHomeSen ACCESS p_DIInvertHomeSen;
	p_bInverterRemoteSen ACCESS p_DIInvertRemoteSen;

	p_eConvStat ACCESS p_ConvStat;
	p_eConvStatus ACCESS p_ConvStatus;
	p_bConvLeftSen ACCESS p_DIConvLftSen;
	p_bConvRightSen ACCESS p_DIConvRgtSen;

	p_eInletShutterStat ACCESS p_Pneu2SenInShutterStat;
	p_eInletShutterStatus ACCESS p_Pneu2SenInShutterStatus;
	p_bInletShutterOpenRs ACCESS p_DIInShutterOpenRS;
	p_bInletShutterCloseRs ACCESS p_DIInShutterCloseRS;

	p_eOutletShutterStat ACCESS p_Pneu2SenOutShutterStat;
	p_eOutletShutterStatus ACCESS p_Pneu2SenOutShutterStatus;
	p_bOutletShutterOpenRs ACCESS p_DIOutShutterOpenRS;
	p_bOutletShutterCloseRs ACCESS p_DIOutShutterCloseRS;

	p_eStopperStat ACCESS p_PneuNoSenStopperStat;
	p_eStopperStatus ACCESS p_PneuNoSenStopperStatus;
	p_bStopperExtended ACCESS p_PneuNoSenStopperExtended;
	p_bStopperRetracted ACCESS p_PneuNoSenStopperRetracted;

	(* Always Change If Project Change *)

END_ACTION
```

#### Act_Link.st - Change By Project
```iecst
(** 2018-12-11 **)
ACTION Act_Link:

END_ACTION
```

#### Cyclic.st - Do Not Change!!!
```iecst
(** 2019-03-22 **)
PROGRAM _CYCLIC

	IF bInitDone = FALSE THEN
		bInitDone	:= TRUE;

		Act_InitLocal;
		Act_InitGlobal;

	ELSIF bInitialDone = FALSE THEN
		IF p_bNtSettingsLoadDone = TRUE THEN
			bInitialDone	:= TRUE;

			Act_Initial;
		END_IF

	ELSE

		Act_RstErr;
		Act_LinkEn;
		Act_Link;
		Act_Background;
		Act_Alarm;

	END_IF

END_PROGRAM
```

#### Act_InitLocal.st - Do Not Change!!!
```iecst
(** 2019-03-25 **)
ACTION Act_InitLocal:

	//Input Reference Link To Local Variable
	p_udiRstErr ACCESS ADR(udiRstErr);
	p_bEn ACCESS ADR(bEn);
	p_bDis ACCESS ADR(bDis);
	p_bRun ACCESS ADR(bRun);
	p_bStop ACCESS ADR(bStop);
	p_bStep ACCESS ADR(bStep);

	p_eInvertStat ACCESS ADR(eInverterStat);
	p_eInvertStatus ACCESS ADR(eInverterStatus);

	p_eConvStat ACCESS ADR(eConvStat);
	p_eConvStatus ACCESS ADR(eConvStatus);

	p_eStopperStat ACCESS ADR(eStopperStat);
	p_eStopperStatus ACCESS ADR(eStopperStatus);

	p_eInletShutterStat ACCESS ADR(eInletShutterStat);
	p_eInletShutterStatus ACCESS ADR(eInletShutterStatus);

	p_eOutletShutterStat ACCESS ADR(eOutletShutterStat);
	p_eOutletShutterStatus ACCESS ADR(eOutletShutterStatus);

	p_bConvLeftSen ACCESS ADR(bConvLeftSen);
	p_bConvRightSen ACCESS ADR(bConvRightSen);

	p_bInletShutterCloseRs ACCESS ADR(bInletShutterCloseRS);
	p_bOutletShutterCloseRs ACCESS ADR(bOutletShutterCloseRS);

	p_sProgNm ACCESS ADR(sProgNm);
	p_bNtSettingsLoadDone ACCESS ADR(bNtSettingsLoadDone);

END_ACTION
```

#### Act_Initial.st - Do Not Change!!!
```iecst
(** 2019-01-20 **)
ACTION Act_Initial:

	//Initial

END_ACTION
```

#### Act_Background.st - Do Not Change!!!
```iecst
(** 2019-01-23 **)
ACTION Act_Background:

	//Reset bPaused
	IF EDGENEG(p_bStop OR p_bStep) THEN
		bPaused	:= FALSE;
	END_IF

	IF eStatus <> Error AND p_bRun = TRUE THEN
		IF (p_bEn = TRUE) AND (p_bDis = FALSE) THEN
			Act_OpsRun;
		ELSE
			bPaused	:= p_bStop OR p_bStep;
		END_IF

		IF EDGEPOS(p_bEn = FALSE OR p_bDis = TRUE) THEN
			Act_OpsRst;
		END_IF

	ELSIF eStatus <> Error THEN
		sStepTxt	:= 'Stop';
	ELSE
		sStepTxt	:= 'Error';
	END_IF

	//Reset
	IF EDGENEG(p_bRun) OR EDGEPOS(eStatus = Error) THEN
		Act_OpsInitial;
		Act_OpsRst;
	END_IF

	//Reset Error
	IF (eStatus = Error) AND bRstErr THEN
		eStatus		:= Idle;
		udiStatus	:= 0;
	END_IF

END_ACTION
```

#### Act_Alarm.st - Do Not Change!!!
```iecst
(** 2019-03-25 **)
ACTION Act_Alarm:

	//Error
	IF EDGEPOS(eStatus = Error) THEN

		tyAlmData.sProgNm		:= p_sProgNm;
		tyAlmData.udiCode		:= udiStatus;
		tyAlmData.eSeverity		:= AlmSeverityError;
		tyAlmData.udiRunTime	:= tyAlmData.udiRunTime + 1;

		//Get Error Message
		IF tyAlmData.udiCode < 10000 OR tyAlmData.udiCode > 10099 THEN
			tyAlmData.sAlmMsg	:= 'Unknown';
			tyAlmData.sRcyMsg	:= 'Unknown';
		ELSE
			tyAlmData.sAlmMsg	:= a_tyAlmText[tyAlmData.udiCode].sAlmText;
			tyAlmData.sRcyMsg	:= a_tyAlmText[tyAlmData.udiCode].sRcyText;
		END_IF

	ELSIF bRstErr AND (tyAlmData.udiCode <> 0) THEN

		tyAlmData.udiCode		:= 0;
		tyAlmData.eSeverity		:= AlmSeverityNA;
		tyAlmData.sAlmMsg		:= '';
		tyAlmData.sRcyMsg		:= '';

	END_IF

END_ACTION
```

#### Package Logical/Simulation/SimuInv/Sequence - Do Not Change!!!

#### Act_OpsInitial.st - Do Not Change!!!
```iecst
(** 2019-01-16 **)
ACTION Act_OpsInitial:

	IF p_bInletShutterPrep OR p_bOutletShutterPrep THEN
		eSimuInvGotoStep	:= SimuInvStepInitShutterCls;
	ELSE
		eSimuInvGotoStep	:= SimuInvStepChkCondition;
	END_IF

	eSimuInvStep		:= SimuInvStepNA;

END_ACTION
```
